REGION Network 14: таймер выключения частотника
   #tmrErrOffUZ(IN := NOT #qUZ AND #iWorkUZ, PT := #tStopPU_FC);   // TON
   IF #Ack OR #PU1.ack.%X5 THEN
       #errOff_UZ_PU1 := FALSE;   // RS flip-flop
   END_IF;
   IF #tmrErrOffUZ.Q THEN #errOff_UZ_PU1 := TRUE; END_IF;
   #PU1.st.%X5 := #errOff_UZ_PU1;
   IF #Ack OR #PU2.ack.%X5 THEN
       #errOff_UZ_PU2 := FALSE;   // RS flip-flop
   END_IF;
   IF #tmrErrOffUZ.Q THEN #errOff_UZ_PU2 := TRUE; END_IF;
   #PU2.st.%X5 := #errOff_UZ_PU2;
END_REGION

REGION Network 15: таймер включения контактора PU1
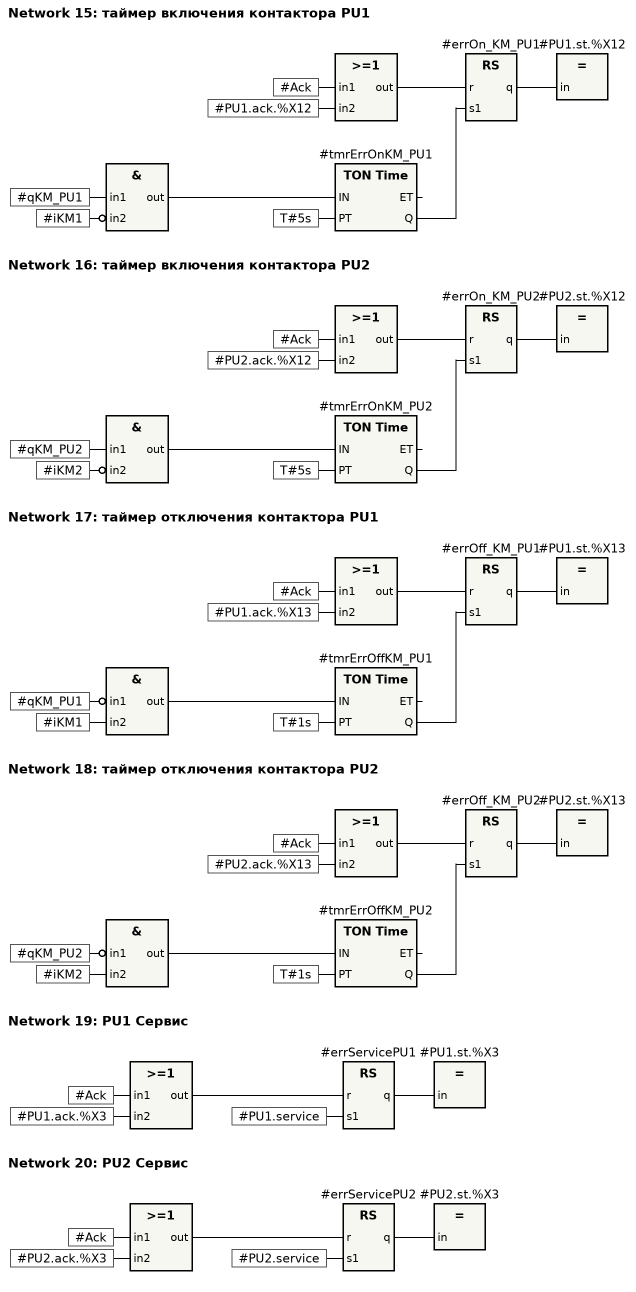
   #tmrErrOnKM_PU1(IN := #qKM_PU1 AND NOT #iKM1, PT := T#5s);   // TON
   IF #Ack OR #PU1.ack.%X12 THEN
       #errOn_KM_PU1 := FALSE;   // RS flip-flop
   END_IF;
   IF #tmrErrOnKM_PU1.Q THEN #errOn_KM_PU1 := TRUE; END_IF;
   #PU1.st.%X12 := #errOn_KM_PU1;
END_REGION

REGION Network 16: таймер включения контактора PU2
   #tmrErrOnKM_PU2(IN := #qKM_PU2 AND NOT #iKM2, PT := T#5s);   // TON
   IF #Ack OR #PU2.ack.%X12 THEN
       #errOn_KM_PU2 := FALSE;   // RS flip-flop
   END_IF;
   IF #tmrErrOnKM_PU2.Q THEN #errOn_KM_PU2 := TRUE; END_IF;
   #PU2.st.%X12 := #errOn_KM_PU2;
END_REGION

REGION Network 17: таймер отключения контактора PU1
   #tmrErrOffKM_PU1(IN := NOT #qKM_PU1 AND #iKM1, PT := T#1s);   // TON
   IF #Ack OR #PU1.ack.%X13 THEN
       #errOff_KM_PU1 := FALSE;   // RS flip-flop
   END_IF;
   IF #tmrErrOffKM_PU1.Q THEN #errOff_KM_PU1 := TRUE; END_IF;
   #PU1.st.%X13 := #errOff_KM_PU1;
END_REGION

REGION Network 18: таймер отключения контактора PU2
   #tmrErrOffKM_PU2(IN := NOT #qKM_PU2 AND #iKM2, PT := T#1s);   // TON
   IF #Ack OR #PU2.ack.%X13 THEN
       #errOff_KM_PU2 := FALSE;   // RS flip-flop
   END_IF;
   IF #tmrErrOffKM_PU2.Q THEN #errOff_KM_PU2 := TRUE; END_IF;
   #PU2.st.%X13 := #errOff_KM_PU2;
END_REGION

REGION Network 19: PU1 Сервис
   IF #Ack OR #PU1.ack.%X3 THEN
       #errServicePU1 := FALSE;   // RS flip-flop
   END_IF;
   IF #PU1.service THEN #errServicePU1 := TRUE; END_IF;
   #PU1.st.%X3 := #errServicePU1;
END_REGION

REGION Network 20: PU2 Сервис
   IF #Ack OR #PU2.ack.%X3 THEN
       #errServicePU2 := FALSE;   // RS flip-flop
   END_IF;
   IF #PU2.service THEN #errServicePU2 := TRUE; END_IF;
   #PU2.st.%X3 := #errServicePU2;
END_REGION

REGION Network 21: Сборная ошибка РU1
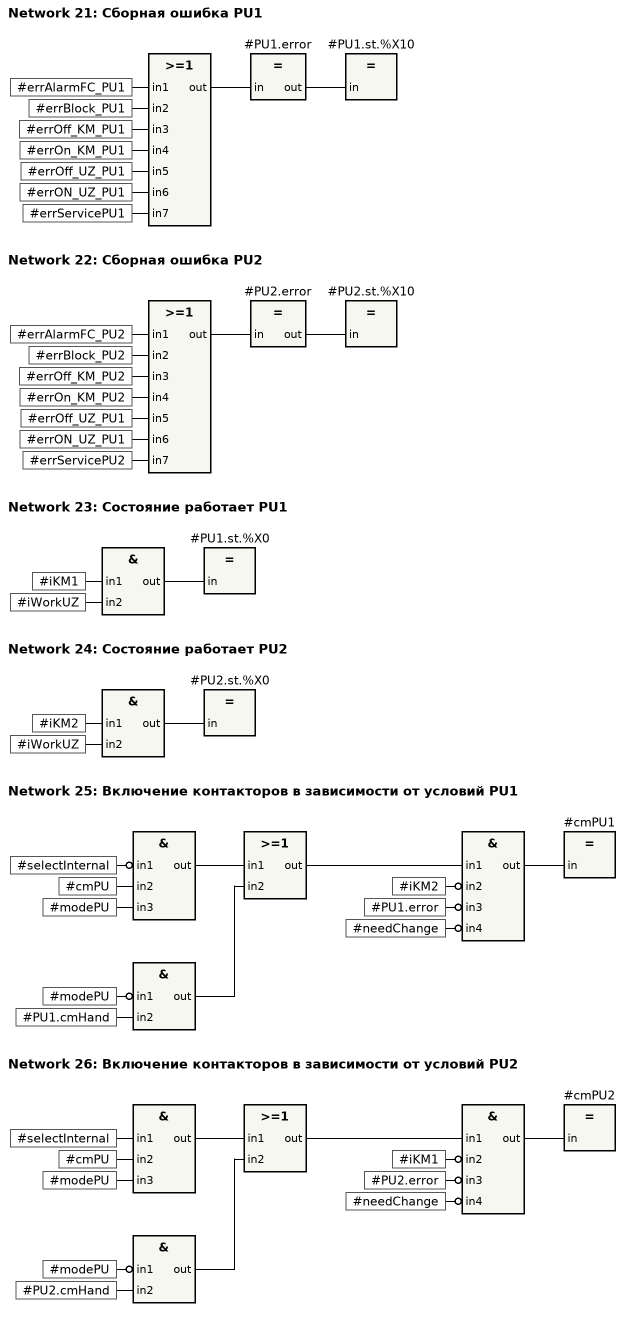
   #PU1.error := #errAlarmFC_PU1 OR #errBlock_PU1 OR #errOff_KM_PU1 OR #errOn_KM_PU1 OR #errOff_UZ_PU1 OR #errON_UZ_PU1 OR #errServicePU1;
   #PU1.st.%X10 := #PU1.error;
END_REGION

REGION Network 22: Сборная ошибка РU2
   #PU2.error := #errAlarmFC_PU2 OR #errBlock_PU2 OR #errOff_KM_PU2 OR #errOn_KM_PU2 OR #errOff_UZ_PU1 OR #errON_UZ_PU1 OR #errServicePU2;
   #PU2.st.%X10 := #PU2.error;
END_REGION

REGION Network 23: Состояние работает PU1
   #PU1.st.%X0 := #iKM1 AND #iWorkUZ;
END_REGION

REGION Network 24: Состояние работает PU2
   #PU2.st.%X0 := #iKM2 AND #iWorkUZ;
END_REGION

REGION Network 25: Включение контакторов в зависимости от условий PU1
   #cmPU1 := ((NOT #selectInternal AND #cmPU AND #modePU) OR (NOT #modePU AND #PU1.cmHand)) AND NOT #iKM2 AND NOT #PU1.error AND NOT #needChange;
END_REGION

REGION Network 26: Включение контакторов в зависимости от условий PU2
   #cmPU2 := ((#selectInternal AND #cmPU AND #modePU) OR (NOT #modePU AND #PU2.cmHand)) AND NOT #iKM1 AND NOT #PU2.error AND NOT #needChange;
END_REGION

REGION Network 27: Rонтактор первого насоса - СТОП
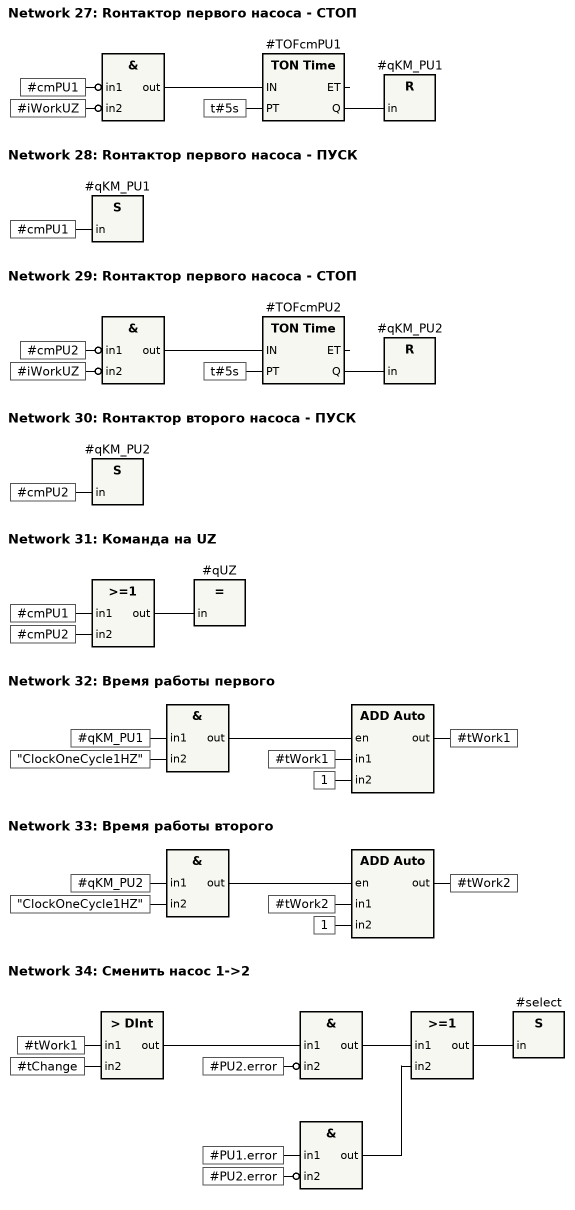
   #TOFcmPU1(IN := NOT #cmPU1 AND NOT #iWorkUZ, PT := t#5s);   // TON
   IF #TOFcmPU1.Q THEN #qKM_PU1 := FALSE; END_IF;
END_REGION

REGION Network 28: Rонтактор первого насоса - ПУСК
   IF #cmPU1 THEN #qKM_PU1 := TRUE; END_IF;
END_REGION

REGION Network 29: Rонтактор первого насоса - СТОП
   #TOFcmPU2(IN := NOT #cmPU2 AND NOT #iWorkUZ, PT := t#5s);   // TON
   IF #TOFcmPU2.Q THEN #qKM_PU2 := FALSE; END_IF;
END_REGION

REGION Network 30: Rонтактор второго насоса - ПУСК
   IF #cmPU2 THEN #qKM_PU2 := TRUE; END_IF;
END_REGION

REGION Network 31: Команда на UZ
   #qUZ := #cmPU1 OR #cmPU2;
END_REGION

REGION Network 32: Время работы первого
   IF #qKM_PU1 AND "ClockOneCycle1HZ" THEN #tWork1 := #tWork1 + 1; END_IF;
END_REGION

REGION Network 33: Время работы второго
   IF #qKM_PU2 AND "ClockOneCycle1HZ" THEN #tWork2 := #tWork2 + 1; END_IF;
END_REGION

REGION Network 34: Сменить насос 1->2
   IF ((#tWork1 > #tChange) AND NOT #PU2.error) OR (#PU1.error AND NOT #PU2.error) THEN
       #select := TRUE;
   END_IF;
END_REGION

REGION Network 35: Сменить насос 2->1
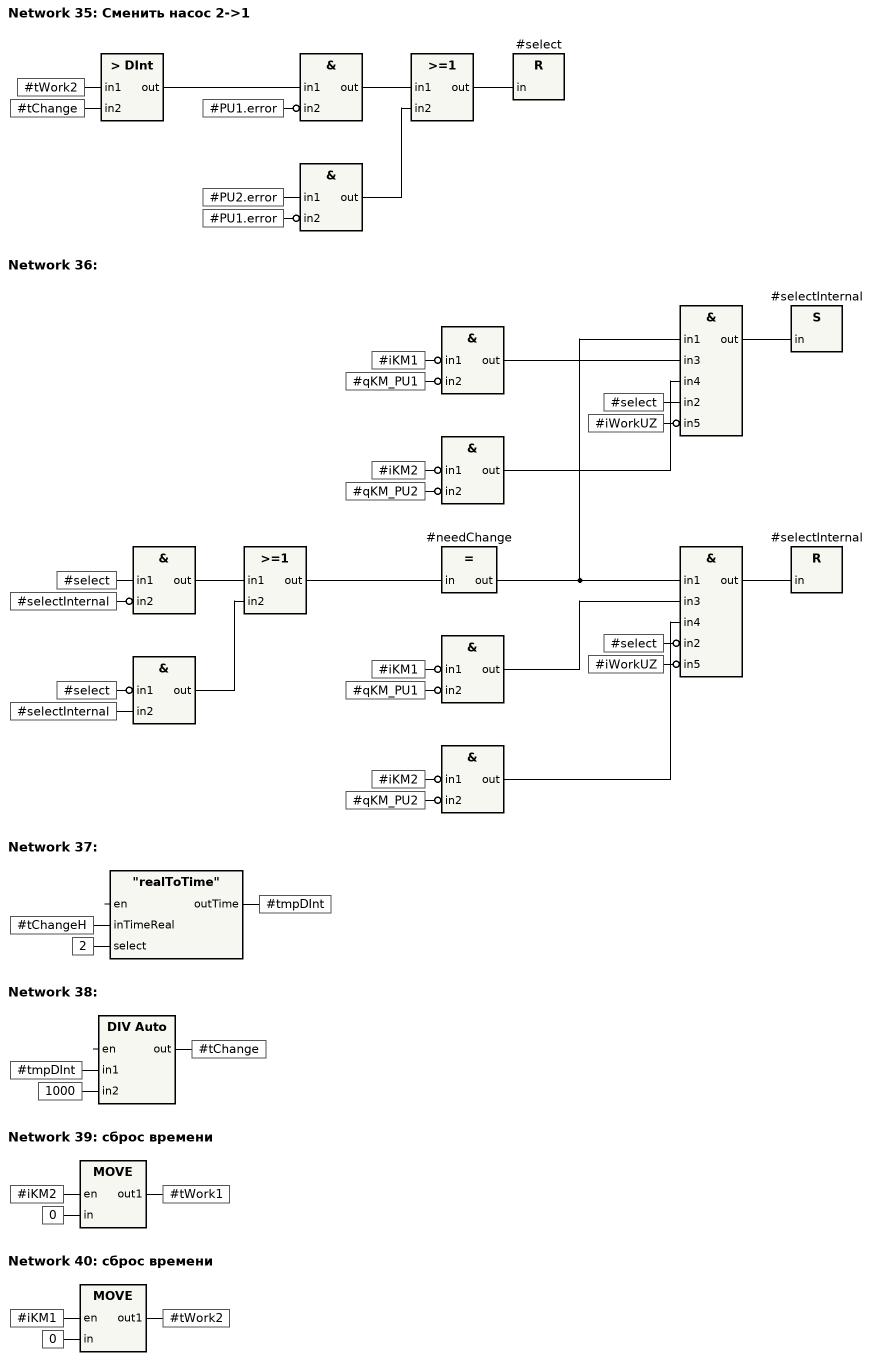
   IF ((#tWork2 > #tChange) AND NOT #PU1.error) OR (#PU2.error AND NOT #PU1.error) THEN
       #select := FALSE;
   END_IF;
END_REGION

REGION Network 36
   #needChange := (#select AND NOT #selectInternal) OR (NOT #select AND #selectInternal);
   IF #needChange AND NOT #iKM1 AND NOT #qKM_PU1 AND NOT #iKM2 AND NOT #qKM_PU2 AND #select AND NOT #iWorkUZ THEN
       #selectInternal := TRUE;
   END_IF;
   IF #needChange AND NOT #iKM1 AND NOT #qKM_PU1 AND NOT #iKM2 AND NOT #qKM_PU2 AND NOT #select AND NOT #iWorkUZ THEN
       #selectInternal := FALSE;
   END_IF;
END_REGION

REGION Network 37
   "realToTime"(inTimeReal := #tChangeH, select := 2, outTime => #tmpDInt);
END_REGION

REGION Network 38
   #tChange := #tmpDInt / 1000;
END_REGION

REGION Network 39: сброс времени
   IF #iKM2 THEN #tWork1 := 0; END_IF;
END_REGION

REGION Network 40: сброс времени
   IF #iKM1 THEN #tWork2 := 0; END_IF;
END_REGION

REGION Network 41: сброс ручных команд - PU1
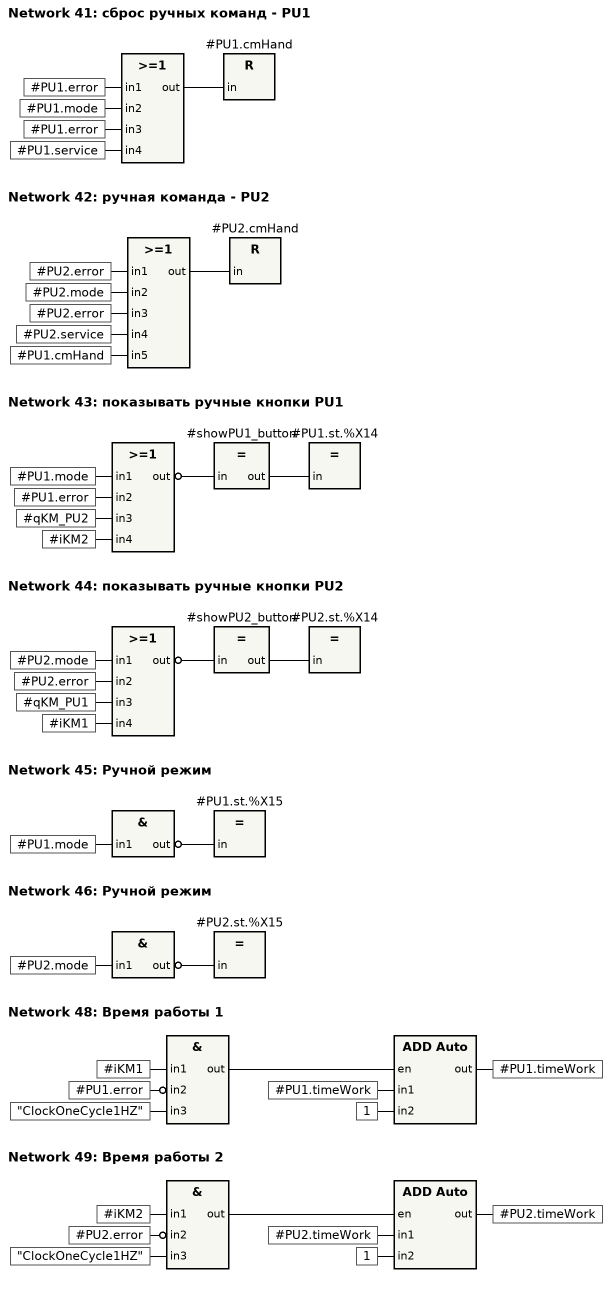
   IF #PU1.error OR #PU1.mode OR #PU1.error OR #PU1.service THEN #PU1.cmHand := FALSE; END_IF;
END_REGION

REGION Network 42: ручная команда - PU2
   IF #PU2.error OR #PU2.mode OR #PU2.error OR #PU2.service OR #PU1.cmHand THEN #PU2.cmHand := FALSE; END_IF;
END_REGION

REGION Network 43: показывать ручные кнопки PU1
   #showPU1_button := NOT (#PU1.mode OR #PU1.error OR #qKM_PU2 OR #iKM2);
   #PU1.st.%X14 := #showPU1_button;
END_REGION

REGION Network 44: показывать ручные кнопки PU2
   #showPU2_button := NOT (#PU2.mode OR #PU2.error OR #qKM_PU1 OR #iKM1);
   #PU2.st.%X14 := #showPU2_button;
END_REGION

REGION Network 45: Ручной режим
   #PU1.st.%X15 := NOT #PU1.mode;
END_REGION

REGION Network 46: Ручной режим
   #PU2.st.%X15 := NOT #PU2.mode;
END_REGION

REGION Network 47 (SCL): Сброс битов Ack
   IF NOT #PU1.st.%X0 AND #PU1.ack.%X0 THEN
       #PU1.ack.%X0 := 0;
   END_IF;
   IF NOT #PU1.st.%X1 AND #PU1.ack.%X1 THEN
       #PU1.ack.%X1 := 0;
   END_IF;
   IF NOT #PU1.st.%X2 AND #PU1.ack.%X2 THEN
       #PU1.ack.%X2 := 0;
   END_IF;
   IF NOT #PU1.st.%X3 AND #PU1.ack.%X3 THEN
       #PU1.ack.%X3 := 0;
   END_IF;
   IF NOT #PU1.st.%X4 AND #PU1.ack.%X4 THEN
       #PU1.ack.%X4 := 0;
   END_IF;
   IF NOT #PU1.st.%X5 AND #PU1.ack.%X5 THEN
       #PU1.ack.%X5 := 0;
   END_IF;
   IF NOT #PU1.st.%X6 AND #PU1.ack.%X6 THEN
       #PU1.ack.%X6 := 0;
   END_IF;
   IF NOT #PU1.st.%X7 AND #PU1.ack.%X7 THEN
       #PU1.ack.%X7 := 0;
   END_IF;
   IF NOT #PU1.st.%X8 AND #PU1.ack.%X8 THEN
       #PU1.ack.%X8 := 0;
   END_IF;
   IF NOT #PU1.st.%X9 AND #PU1.ack.%X9 THEN
       #PU1.ack.%X9 := 0;
   END_IF;
   IF NOT #PU1.st.%X10 AND #PU1.ack.%X10 THEN
       #PU1.ack.%X10 := 0;
   END_IF;
   IF NOT #PU1.st.%X11 AND #PU1.ack.%X11 THEN
       #PU1.ack.%X11 := 0;
   END_IF;
   IF NOT #PU1.st.%X12 AND #PU1.ack.%X12 THEN
       #PU1.ack.%X12 := 0;
   END_IF;
   IF NOT #PU1.st.%X13 AND #PU1.ack.%X13 THEN
       #PU1.ack.%X13 := 0;
   END_IF;
   IF NOT #PU1.st.%X14 AND #PU1.ack.%X14 THEN
       #PU1.ack.%X14 := 0;
   END_IF;
   IF NOT #PU1.st.%X15 AND #PU1.ack.%X15 THEN
       #PU1.ack.%X15 := 0;
   END_IF;
   IF NOT #PU2.st.%X0 AND #PU2.ack.%X0 THEN
       #PU2.ack.%X0 := 0;
   END_IF;
   IF NOT #PU2.st.%X1 AND #PU2.ack.%X1 THEN
       #PU2.ack.%X1 := 0;
   END_IF;
   IF NOT #PU2.st.%X2 AND #PU2.ack.%X2 THEN
       #PU2.ack.%X2 := 0;
   END_IF;
   IF NOT #PU2.st.%X3 AND #PU2.ack.%X3 THEN
       #PU2.ack.%X3 := 0;
   END_IF;
   IF NOT #PU2.st.%X4 AND #PU2.ack.%X4 THEN
       #PU2.ack.%X4 := 0;
   END_IF;
   IF NOT #PU2.st.%X5 AND #PU2.ack.%X5 THEN
       #PU2.ack.%X5 := 0;
   END_IF;
   IF NOT #PU2.st.%X6 AND #PU2.ack.%X6 THEN
       #PU2.ack.%X6 := 0;
   END_IF;
   IF NOT #PU2.st.%X7 AND #PU2.ack.%X7 THEN
       #PU2.ack.%X7 := 0;
   END_IF;
   IF NOT #PU2.st.%X8 AND #PU2.ack.%X8 THEN
       #PU2.ack.%X8 := 0;
   END_IF;
   IF NOT #PU2.st.%X9 AND #PU2.ack.%X9 THEN
       #PU2.ack.%X9 := 0;
   END_IF;
   IF NOT #PU2.st.%X10 AND #PU2.ack.%X10 THEN
       #PU2.ack.%X10 := 0;
   END_IF;
   IF NOT #PU2.st.%X11 AND #PU2.ack.%X11 THEN
       #PU2.ack.%X11 := 0;
   END_IF;
   IF NOT #PU2.st.%X12 AND #PU2.ack.%X12 THEN
       #PU2.ack.%X12 := 0;
   END_IF;
   IF NOT #PU2.st.%X13 AND #PU2.ack.%X13 THEN
       #PU2.ack.%X13 := 0;
   END_IF;
   IF NOT #PU2.st.%X14 AND #PU2.ack.%X14 THEN
       #PU2.ack.%X14 := 0;
   END_IF;
   IF NOT #PU2.st.%X15 AND #PU2.ack.%X15 THEN
       #PU2.ack.%X15 := 0;
   END_IF;
END_REGION

REGION Network 48: Время работы 1
   IF #iKM1 AND NOT #PU1.error AND "ClockOneCycle1HZ" THEN #PU1.timeWork := #PU1.timeWork + 1; END_IF;
END_REGION

REGION Network 49: Время работы 2
   IF #iKM2 AND NOT #PU2.error AND "ClockOneCycle1HZ" THEN #PU2.timeWork := #PU2.timeWork + 1; END_IF;
END_REGION

REGION Network 50: Сброс 1
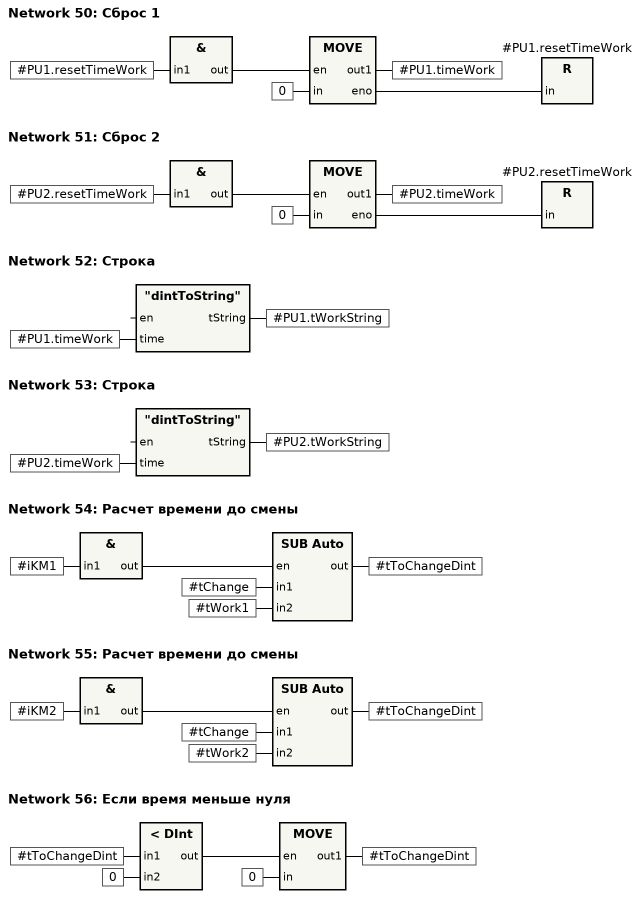
   IF #PU1.resetTimeWork THEN
       #PU1.timeWork := 0;
       #PU1.resetTimeWork := FALSE;
   END_IF;
END_REGION

REGION Network 51: Сброс 2
   IF #PU2.resetTimeWork THEN
       #PU2.timeWork := 0;
       #PU2.resetTimeWork := FALSE;
   END_IF;
END_REGION

REGION Network 52: Строка
   "dintToString"("time" := #PU1.timeWork, tString => #PU1.tWorkString);
END_REGION

REGION Network 53: Строка
   "dintToString"("time" := #PU2.timeWork, tString => #PU2.tWorkString);
END_REGION

REGION Network 54: Расчет времени до смены
   IF #iKM1 THEN #tToChangeDint := #tChange - #tWork1; END_IF;
END_REGION

REGION Network 55: Расчет времени до смены
   IF #iKM2 THEN #tToChangeDint := #tChange - #tWork2; END_IF;
END_REGION

REGION Network 56: Если время меньше нуля
   IF #tToChangeDint < 0 THEN #tToChangeDint := 0; END_IF;
END_REGION

REGION Network 57 (SCL): Сек -> час
   #tToChangeRealHour := DINT_TO_REAL(#tToChangeDint) / 3600.0;
END_REGION
END_FUNCTION_BLOCK

FUNCTION "intToTime" : Void
{ S7_Optimized_Access := 'TRUE' }
VERSION : 0.1
   VAR_INPUT 
      intTime : Int;
      select : Int;   // 0-sec, 1-min,2-hour
   END_VAR

   VAR_OUTPUT 
      tOut : Time;
   END_VAR


BEGIN
	CASE #select OF
	    0:
	        #tOut := DINT_TO_TIME(INT_TO_DINT(#intTime) * 1000);
	    1:
	        #tOut := DINT_TO_TIME(INT_TO_DINT(#intTime)* 60000);
	    2:
	        #tOut := DINT_TO_TIME(INT_TO_DINT(#intTime) * 3600000);
	    ELSE  // Statement section ELSE
	        #tOut := t#0s;
	END_CASE;
END_FUNCTION

FUNCTION "bitToWord" : Void   // FC5, LAD
{ S7_Optimized_Access := 'TRUE' }
VERSION : 0.1
// stored: AutoNumber true, IsIECCheckEnabled false, SetENOAutomatically false, UDAEnableTagReadback false
   VAR_INPUT
      inBit0 : Bool;
      inBit1 : Bool;
      inBit2 : Bool;
      inBit3 : Bool;
      inBit4 : Bool;
      inBit5 : Bool;
      inBit6 : Bool;
      inBit7 : Bool;
      inBit8 : Bool;
      inBit9 : Bool;
      inBit10 : Bool;
      inBit11 : Bool;
      inBit12 : Bool;
      inBit13 : Bool;
      inBit14 : Bool;
      inBit15 : Bool;
   END_VAR
   VAR_OUTPUT
      outWord : Word;
   END_VAR
BEGIN

REGION Network 1
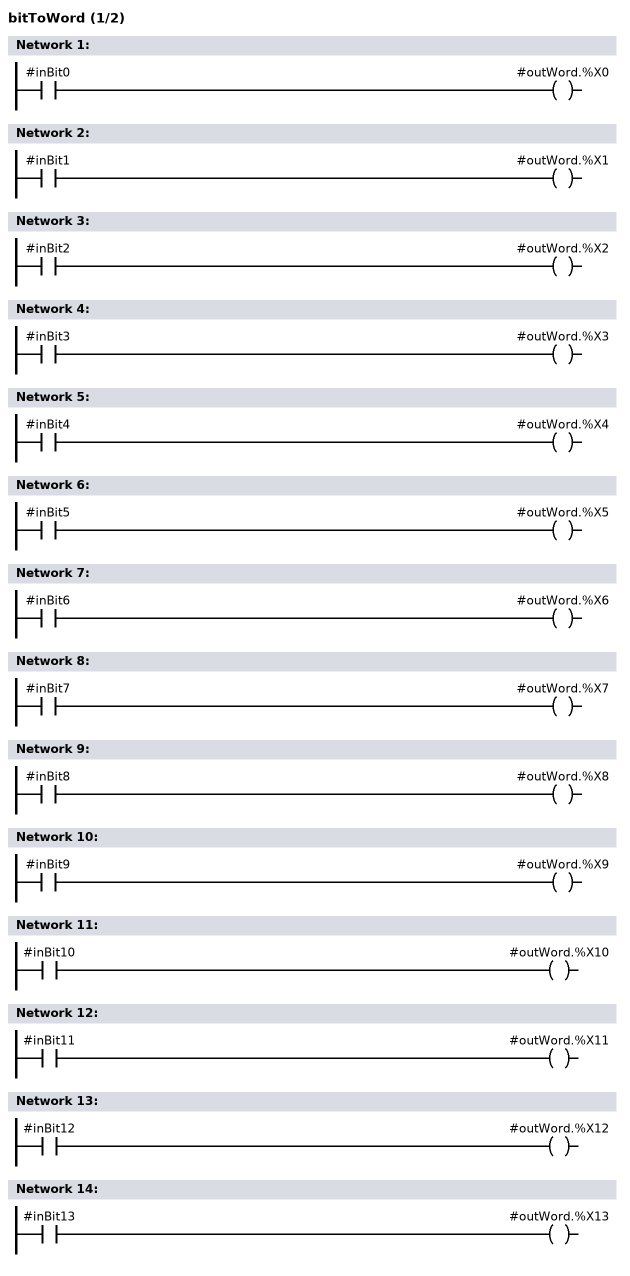
   RUNG wire#powerrail
      Contact( #inBit0 )
      Coil( #outWord.%X0 )
   END_RUNG
   // the same network as SCL:
   #outWord.%X0 := #inBit0;
END_REGION

REGION Network 2
   RUNG wire#powerrail
      Contact( #inBit1 )
      Coil( #outWord.%X1 )
   END_RUNG
   // the same network as SCL:
   #outWord.%X1 := #inBit1;
END_REGION

REGION Network 3
   RUNG wire#powerrail
      Contact( #inBit2 )
      Coil( #outWord.%X2 )
   END_RUNG
   // the same network as SCL:
   #outWord.%X2 := #inBit2;
END_REGION

REGION Network 4
   RUNG wire#powerrail
      Contact( #inBit3 )
      Coil( #outWord.%X3 )
   END_RUNG
   // the same network as SCL:
   #outWord.%X3 := #inBit3;
END_REGION

REGION Network 5
   RUNG wire#powerrail
      Contact( #inBit4 )
      Coil( #outWord.%X4 )
   END_RUNG
   // the same network as SCL:
   #outWord.%X4 := #inBit4;
END_REGION

REGION Network 6
   RUNG wire#powerrail
      Contact( #inBit5 )
      Coil( #outWord.%X5 )
   END_RUNG
   // the same network as SCL:
   #outWord.%X5 := #inBit5;
END_REGION

REGION Network 7
   RUNG wire#powerrail
      Contact( #inBit6 )
      Coil( #outWord.%X6 )
   END_RUNG
   // the same network as SCL:
   #outWord.%X6 := #inBit6;
END_REGION

REGION Network 8
   RUNG wire#powerrail
      Contact( #inBit7 )
      Coil( #outWord.%X7 )
   END_RUNG
   // the same network as SCL:
   #outWord.%X7 := #inBit7;
END_REGION

REGION Network 9
   RUNG wire#powerrail
      Contact( #inBit8 )
      Coil( #outWord.%X8 )
   END_RUNG
   // the same network as SCL:
   #outWord.%X8 := #inBit8;
END_REGION

REGION Network 10
   RUNG wire#powerrail
      Contact( #inBit9 )
      Coil( #outWord.%X9 )
   END_RUNG
   // the same network as SCL:
   #outWord.%X9 := #inBit9;
END_REGION

REGION Network 11
   RUNG wire#powerrail
      Contact( #inBit10 )
      Coil( #outWord.%X10 )
   END_RUNG
   // the same network as SCL:
   #outWord.%X10 := #inBit10;
END_REGION

REGION Network 12
   RUNG wire#powerrail
      Contact( #inBit11 )
      Coil( #outWord.%X11 )
   END_RUNG
   // the same network as SCL:
   #outWord.%X11 := #inBit11;
END_REGION

REGION Network 13
   RUNG wire#powerrail
      Contact( #inBit12 )
      Coil( #outWord.%X12 )
   END_RUNG
   // the same network as SCL:
   #outWord.%X12 := #inBit12;
END_REGION

REGION Network 14
   RUNG wire#powerrail
      Contact( #inBit13 )
      Coil( #outWord.%X13 )
   END_RUNG
   // the same network as SCL:
   #outWord.%X13 := #inBit13;
END_REGION

REGION Network 15
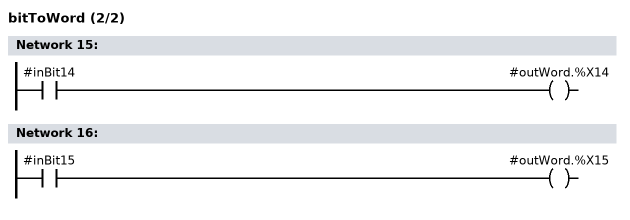
   RUNG wire#powerrail
      Contact( #inBit14 )
      Coil( #outWord.%X14 )
   END_RUNG
   // the same network as SCL:
   #outWord.%X14 := #inBit14;
END_REGION

REGION Network 16
   RUNG wire#powerrail
      Contact( #inBit15 )
      Coil( #outWord.%X15 )
   END_RUNG
   // the same network as SCL:
   #outWord.%X15 := #inBit15;
END_REGION
END_FUNCTION

FUNCTION "realToTime" : Void
{ S7_Optimized_Access := 'TRUE' }
VERSION : 0.1
   VAR_INPUT 
      inTimeReal : Real;
      select : Int;   // 0-секунды, 1-минуты, 2-часы
   END_VAR

   VAR_OUTPUT 
      outTime : Time;
   END_VAR


BEGIN
	CASE #select OF
	    0:
	        #outTime := DINT_TO_TIME(REAL_TO_DINT(#inTimeReal * 1000.0));
	    1:
	        #outTime := DINT_TO_TIME(REAL_TO_DINT(#inTimeReal * 60000.0));
	    2:
	        #outTime := DINT_TO_TIME(REAL_TO_DINT(#inTimeReal * 1000.0) * 3600);
	    ELSE  // Statement section ELSE
	        #outTime := t#0s;
	END_CASE;
	
END_FUNCTION

FUNCTION "dintToString" : Void
{ S7_Optimized_Access := 'TRUE' }
VERSION : 0.1
   VAR_INPUT 
      "time" : UDInt;
   END_VAR

   VAR_OUTPUT 
      tString : String;
   END_VAR

   VAR_TEMP 
      tDInt : UDInt;
      size : USInt;
      pos : USInt;
      day : DInt;
      h : DInt;
      m : DInt;
      s : DInt;
   END_VAR


BEGIN
	#tDInt := #time;
	
	//сбор строки
	#day := #tDInt / 86400;
	#h := (#tDInt MOD 86400) / 3600;
	#m := (#tDInt MOD 3600) / 60;
	#s := #tDInt MOD 60;
	#tString := '00000:00:00:00';
	
	VAL_STRG(IN := #day,
	         SIZE := 5,
	         PREC := 0,
	         FORMAT := 1,
	         P := 1,
	         OUT => #tString);
	
	IF #h < 10 THEN
	    #size := 1;
	    #pos := 8;
	ELSE
	    #size := 2;
	    #pos := 7;
	END_IF;
	
	VAL_STRG(IN := #h,
	         SIZE := #size,
	         PREC := 0,
	         FORMAT := 1,
	         P := #pos,
	         OUT => #tString);
	
	IF #m < 10 THEN
	    #size := 1;
	    #pos := 11;
	ELSE
	    #size := 2;
	    #pos := 10;
	END_IF;
	
	VAL_STRG(IN := #m,
	         SIZE := #size,
	         PREC := 0,
	         FORMAT := 1,
	         P := #pos,
	         OUT => #tString);
	IF #s < 10 THEN
	    #size := 1;
	    #pos := 14;
	ELSE
	    #size := 2;
	    #pos := 13;
	END_IF;
	VAL_STRG(IN := #s,
	         SIZE := #size,
	         PREC := 0,
	         FORMAT := 1,
	         P := #pos,
	         OUT => #tString);
END_FUNCTION

FUNCTION_BLOCK "noPulseTOF"   // FB15, FBD
{ S7_Optimized_Access := 'TRUE' }
VERSION : 0.1
// stored: AutoNumber true, IsIECCheckEnabled false, IsRetainMemResEnabled false, MemoryReserve 100, SetENOAutomatically false, UDAEnableTagReadback false
   VAR_INPUT
      pulse : Bool;
      timeSP_sec : Real;
      reset : Bool;
   END_VAR
   VAR_OUTPUT
      out : Bool;
   END_VAR
   VAR
      curTime : Real;
      nTrig : Bool;
      pTirg : Bool;
   END_VAR
   VAR_TEMP   // added for the SCL form of the ladder/FBD networks
      _w1 : Bool;
      _w2 : Bool;
   END_VAR
BEGIN

REGION Network 1: Увеличение времени
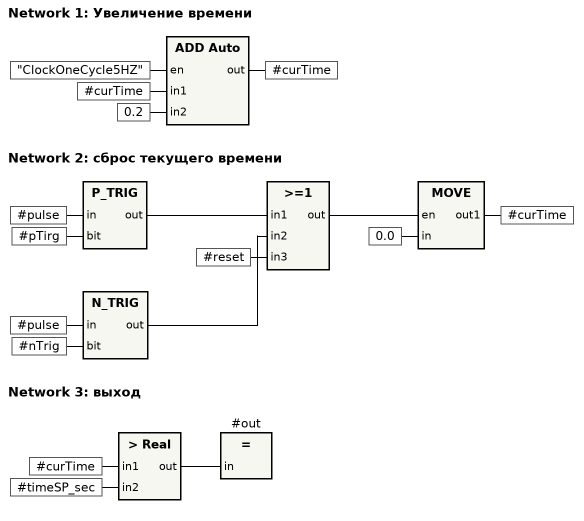
   IF "ClockOneCycle5HZ" THEN #curTime := #curTime + 0.2; END_IF;
END_REGION

REGION Network 2: сброс текущего времени
   #_w1 := #pulse AND NOT #pTirg;   // rising edge
   #pTirg := #pulse;
   #_w2 := NOT #pulse AND #nTrig;   // falling edge
   #nTrig := #pulse;
   IF #_w1 OR #_w2 OR #reset THEN #curTime := 0.0; END_IF;
END_REGION

REGION Network 3: выход
   #out := #curTime > #timeSP_sec;
END_REGION
END_FUNCTION_BLOCK

FUNCTION_BLOCK "sel2pu"   // FB4, FBD
{ S7_Optimized_Access := 'TRUE' }
VERSION : 0.1
// stored: AutoNumber true, IsIECCheckEnabled false, IsRetainMemResEnabled false, MemoryReserve 100, SetENOAutomatically false, UDAEnableTagReadback false
   VAR_INPUT
      cmStart : Bool;
      mode : Bool;
      tChangeHReal : Real;
   END_VAR
   VAR_OUTPUT
      tToChange : Real;
   END_VAR
   VAR_IN_OUT
      PU1 : "Pump";
      PU2 : "Pump";
      select : Bool;
   END_VAR
   VAR
      tWork1 : DInt;
      tWork2 : DInt;
      tChangeDInt : DInt;
   END_VAR
BEGIN

REGION Network 1: Режим работы
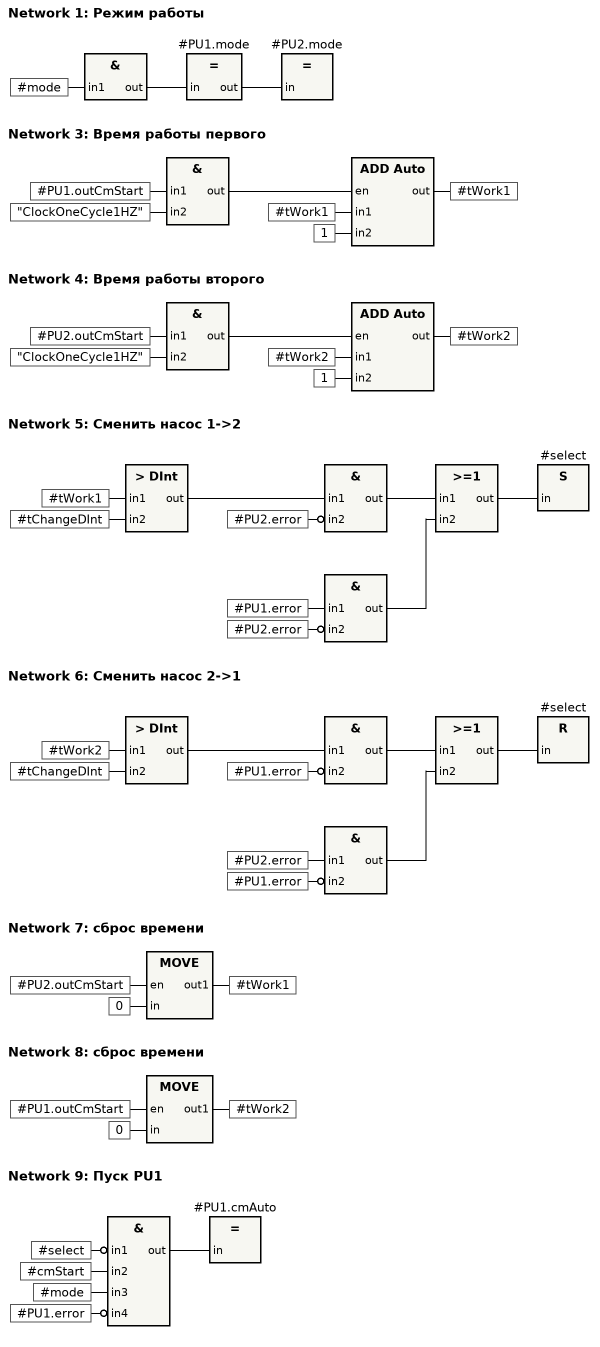
   #PU1.mode := #mode;
   #PU2.mode := #mode;
END_REGION

REGION Network 2 (SCL): Преобразование времен
   #tChangeDInt := REAL_TO_DINT(#tChangeHReal * 3600.0);
END_REGION

REGION Network 3: Время работы первого
   IF #PU1.outCmStart AND "ClockOneCycle1HZ" THEN #tWork1 := #tWork1 + 1; END_IF;
END_REGION

REGION Network 4: Время работы второго
   IF #PU2.outCmStart AND "ClockOneCycle1HZ" THEN #tWork2 := #tWork2 + 1; END_IF;
END_REGION

REGION Network 5: Сменить насос 1->2
   IF ((#tWork1 > #tChangeDInt) AND NOT #PU2.error) OR (#PU1.error AND NOT #PU2.error) THEN
       #select := TRUE;
   END_IF;
END_REGION

REGION Network 6: Сменить насос 2->1
   IF ((#tWork2 > #tChangeDInt) AND NOT #PU1.error) OR (#PU2.error AND NOT #PU1.error) THEN
       #select := FALSE;
   END_IF;
END_REGION

REGION Network 7: сброс времени
   IF #PU2.outCmStart THEN #tWork1 := 0; END_IF;
END_REGION

REGION Network 8: сброс времени
   IF #PU1.outCmStart THEN #tWork2 := 0; END_IF;
END_REGION

REGION Network 9: Пуск PU1
   #PU1.cmAuto := NOT #select AND #cmStart AND #mode AND NOT #PU1.error;
END_REGION

REGION Network 10: Пуск PU2
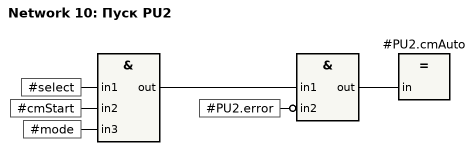
   #PU2.cmAuto := #select AND #cmStart AND #mode AND NOT #PU2.error;
END_REGION
END_FUNCTION_BLOCK

FUNCTION_BLOCK "PumpCntr"   // FB60, LAD
{ S7_Optimized_Access := 'FALSE' }
VERSION : 0.1
// #ST:
// номер бита, часло десятичное
//  0  - стоп 
// 0 1 - работа
// 1 2 - запуск
// 2 4 - остановка
// 3 8 - сервисный режим
// 4 16 - ошибка Пуска
// 5 32 - ошибка Стопа
// 6 64 - ошибка питания
// 7 128 - ошибка частотника (дозатора)
// 8 256 - Блокировка внешняя
// 9 - 512 - нажат аварийный стоп
// 10 -1024 - сборная авария
// 11 2048 - местный режим
// 12 4096
// 13 8192
// 14 16384 1-показывать кнопки ручного управления
// 15 32768 - режим 1-ручной, 0-авто (только для индкатора на скаде)
// stored: AutoNumber false, IsIECCheckEnabled false, SetENOAutomatically false, UDAEnableTagReadback false
   VAR_INPUT
      power : Bool;   // питание устройства 1-ок
      run : Bool;   // 1-работа
      emrStop : Bool;   // Авариный стоп 0-авария, 1-ок
      local : Bool;   // 1-местный режим
      alarmFC : Bool;   // 1-авария
      block1 : Bool;
      block2 : Bool;
      block3 : Bool;
      block4 : Bool;
      block5 : Bool;
      block6 : Bool;
      block7 : Bool;
      block8 : Bool;
   END_VAR
   VAR_OUTPUT
      qStart : Bool;   // пуск
   END_VAR
   VAR_IN_OUT
      dev : "Pump";
   END_VAR
   VAR DB_SPECIFIC
      ErrOC : Bool;   // Признак аварии по закрытию или открытию
      ErrPower : Bool;   // Признак аварии питания
      ErrDis : Bool;   // Признак внешней блокировки
      qON : Bool;   // Выход для управления механизмом
      tmrClosing { S7_SetPoint := 'True'} : TON_TIME;
      tmrOpening { S7_SetPoint := 'True'} : TON_TIME;
      closed : Bool;
      opened : Bool;
      closing : Bool;
      opening : Bool;
      errStart : Bool;
      errStop : Bool;
      errEmrStop : Bool;
      errAlarmFc : Bool;
      errService : Bool;
      errLocal : Bool;
      tStart : Time;
      tStop : Time;
   END_VAR
   VAR
      DpumpAckAlarm_Instance : "PumpAckAlarm";
   END_VAR
   VAR CONSTANT
      ACK_DELAY : Time := T#1s;
   END_VAR
BEGIN

REGION Network 1: Сброс состояния
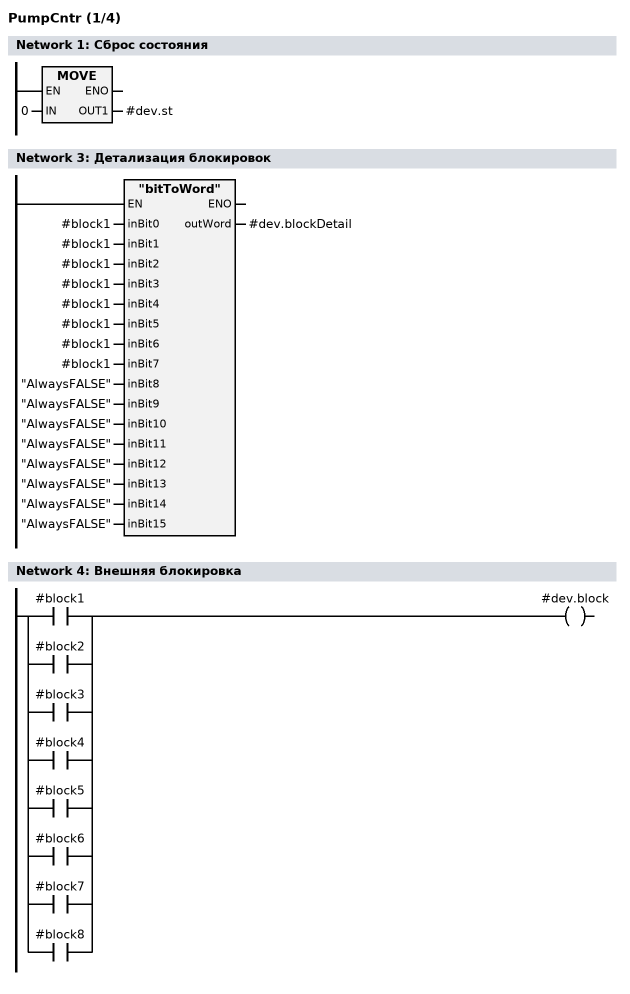
   RUNG wire#powerrail
      { S7_GenerateENO := "TRUE" } Move(in := 0, out1 => #dev.st)
   END_RUNG
   // the same network as SCL:
   #dev.st := 0;
END_REGION

REGION Network 3: Детализация блокировок
   RUNG wire#powerrail
      "bitToWord"(inBit0 := #block1, inBit1 := #block1, inBit2 := #block1, inBit3 := #block1, inBit4 := #block1, inBit5 := #block1, inBit6 := #block1, inBit7 := #block1, inBit8 := "AlwaysFALSE", inBit9 := "AlwaysFALSE", inBit10 := "AlwaysFALSE", inBit11 := "AlwaysFALSE", inBit12 := "AlwaysFALSE", inBit13 := "AlwaysFALSE", inBit14 := "AlwaysFALSE", inBit15 := "AlwaysFALSE", outWord => #dev.blockDetail)
   END_RUNG
   // the same network as SCL:
   "bitToWord"(inBit0 := #block1,
               inBit1 := #block1,
               inBit2 := #block1,
               inBit3 := #block1,
               inBit4 := #block1,
               inBit5 := #block1,
               inBit6 := #block1,
               inBit7 := #block1,
               inBit8 := "AlwaysFALSE",
               inBit9 := "AlwaysFALSE",
               inBit10 := "AlwaysFALSE",
               inBit11 := "AlwaysFALSE",
               inBit12 := "AlwaysFALSE",
               inBit13 := "AlwaysFALSE",
               inBit14 := "AlwaysFALSE",
               inBit15 := "AlwaysFALSE",
               outWord => #dev.blockDetail);
END_REGION

REGION Network 4: Внешняя блокировка
   RUNG wire#powerrail
      Contact( #block1 )
      wire#w1
      Coil( #dev.block )
   END_RUNG
   RUNG wire#powerrail
      Contact( #block2 )
   END_RUNG wire#w1
   RUNG wire#powerrail
      Contact( #block3 )
   END_RUNG wire#w1
   RUNG wire#powerrail
      Contact( #block4 )
   END_RUNG wire#w1
   RUNG wire#powerrail
      Contact( #block5 )
   END_RUNG wire#w1
   RUNG wire#powerrail
      Contact( #block6 )
   END_RUNG wire#w1
   RUNG wire#powerrail
      Contact( #block7 )
   END_RUNG wire#w1
   RUNG wire#powerrail
      Contact( #block8 )
   END_RUNG wire#w1
   // the same network as SCL:
   #dev.block := #block1 OR #block2 OR #block3 OR #block4 OR #block5 OR #block6 OR #block7 OR #block8;
END_REGION

REGION Network 5: Alarms
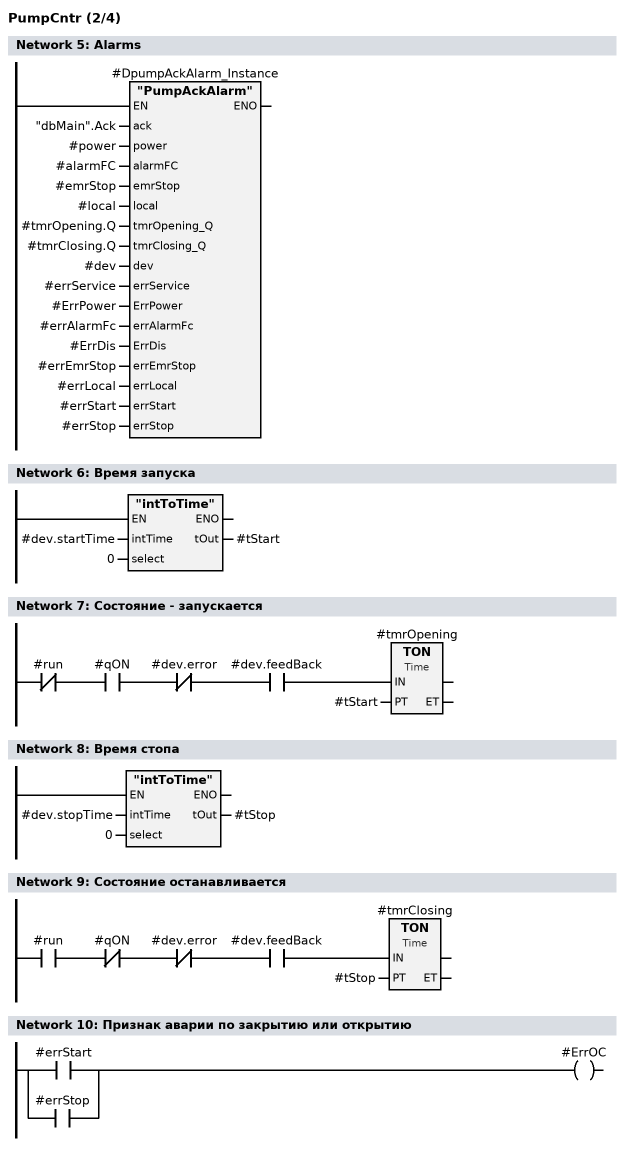
   RUNG wire#powerrail
      #DpumpAckAlarm_Instance(ack := "dbMain".Ack, power := #power, alarmFC := #alarmFC, emrStop := #emrStop, local := #local, tmrOpening_Q := #tmrOpening.Q, tmrClosing_Q := #tmrClosing.Q, dev := #dev, errService := #errService, ErrPower := #ErrPower, errAlarmFc := #errAlarmFc, ErrDis := #ErrDis, errEmrStop := #errEmrStop, errLocal := #errLocal, errStart := #errStart, errStop := #errStop)
   END_RUNG
   // the same network as SCL:
   #DpumpAckAlarm_Instance(ack := "dbMain".Ack,   // "PumpAckAlarm"
                           power := #power,
                           alarmFC := #alarmFC,
                           emrStop := #emrStop,
                           local := #local,
                           tmrOpening_Q := #tmrOpening.Q,
                           tmrClosing_Q := #tmrClosing.Q,
                           dev := #dev,
                           errService := #errService,
                           ErrPower := #ErrPower,
                           errAlarmFc := #errAlarmFc,
                           ErrDis := #ErrDis,
                           errEmrStop := #errEmrStop,
                           errLocal := #errLocal,
                           errStart := #errStart,
                           errStop := #errStop);
END_REGION

REGION Network 6: Время запуска
   RUNG wire#powerrail
      "intToTime"(intTime := #dev.startTime, select := 0, tOut => #tStart)
   END_RUNG
   // the same network as SCL:
   "intToTime"(intTime := #dev.startTime, select := 0, tOut => #tStart);
END_REGION

REGION Network 7: Состояние - запускается
   RUNG wire#powerrail
      I_Contact( #run )
      Contact( #qON )
      I_Contact( #dev.error )
      Contact( #dev.feedBack )
      { S7_Templates := "time_type := Time" } #tmrOpening.TON(pt := #tStart, et =>)
   END_RUNG
   // the same network as SCL:
   #tmrOpening(IN := NOT #run AND #qON AND NOT #dev.error AND #dev.feedBack, PT := #tStart);   // TON
END_REGION

REGION Network 8: Время стопа
   RUNG wire#powerrail
      "intToTime"(intTime := #dev.stopTime, select := 0, tOut => #tStop)
   END_RUNG
   // the same network as SCL:
   "intToTime"(intTime := #dev.stopTime, select := 0, tOut => #tStop);
END_REGION

REGION Network 9: Состояние останавливается
   RUNG wire#powerrail
      Contact( #run )
      I_Contact( #qON )
      I_Contact( #dev.error )
      Contact( #dev.feedBack )
      { S7_Templates := "time_type := Time" } #tmrClosing.TON(pt := #tStop, et =>)
   END_RUNG
   // the same network as SCL:
   #tmrClosing(IN := #run AND NOT #qON AND NOT #dev.error AND #dev.feedBack, PT := #tStop);   // TON
END_REGION

REGION Network 10: Признак аварии по закрытию или открытию
   RUNG wire#powerrail
      Contact( #errStart )
      wire#w1
      Coil( #ErrOC )
   END_RUNG
   RUNG wire#powerrail
      Contact( #errStop )
   END_RUNG wire#w1
   // the same network as SCL:
   #ErrOC := #errStart OR #errStop;
END_REGION

REGION Network 11: Сборная авария
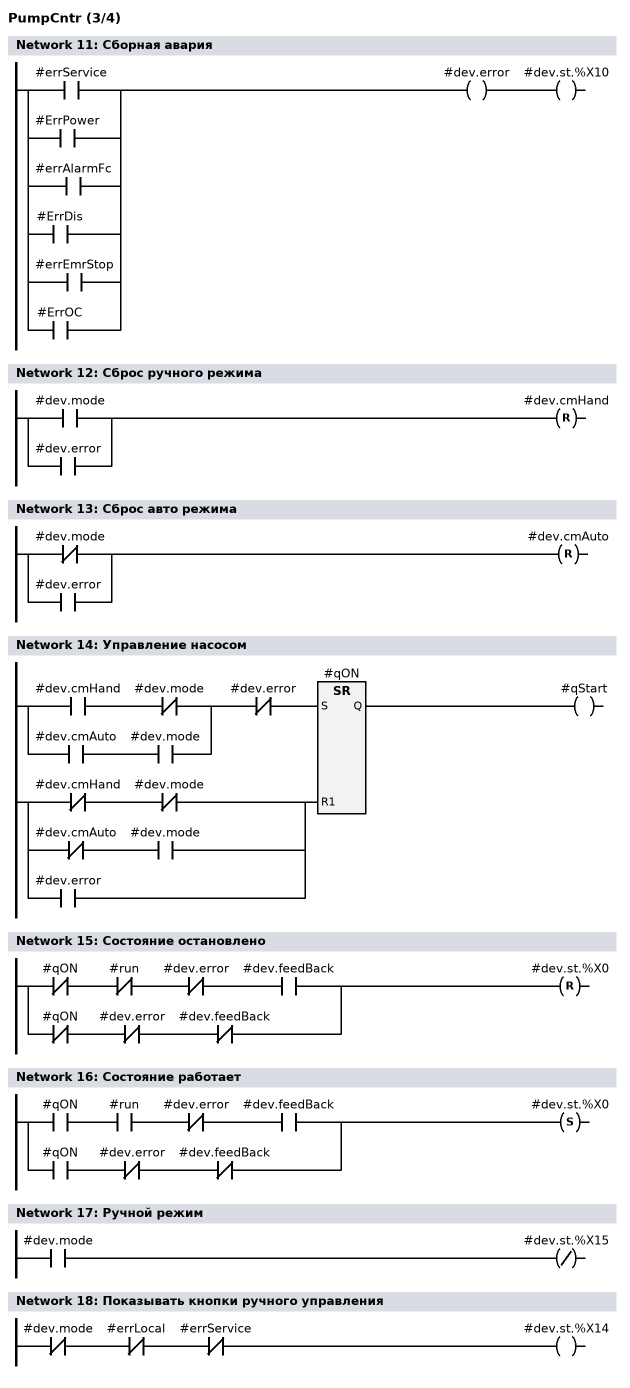
   RUNG wire#powerrail
      Contact( #errService )
      wire#w1
      Coil( #dev.error )
      Coil( #dev.st.%X10 )
   END_RUNG
   RUNG wire#powerrail
      Contact( #ErrPower )
   END_RUNG wire#w1
   RUNG wire#powerrail
      Contact( #errAlarmFc )
   END_RUNG wire#w1
   RUNG wire#powerrail
      Contact( #ErrDis )
   END_RUNG wire#w1
   RUNG wire#powerrail
      Contact( #errEmrStop )
   END_RUNG wire#w1
   RUNG wire#powerrail
      Contact( #ErrOC )
   END_RUNG wire#w1
   // the same network as SCL:
   #dev.error := #errService OR #ErrPower OR #errAlarmFc OR #ErrDis OR #errEmrStop OR #ErrOC;
   #dev.st.%X10 := #dev.error;
END_REGION

REGION Network 12: Сброс ручного режима
   RUNG wire#powerrail
      Contact( #dev.mode )
      wire#w1
      R_Coil( #dev.cmHand )
   END_RUNG
   RUNG wire#powerrail
      Contact( #dev.error )
   END_RUNG wire#w1
   // the same network as SCL:
   IF #dev.mode OR #dev.error THEN #dev.cmHand := FALSE; END_IF;
END_REGION

REGION Network 13: Сброс авто режима
   RUNG wire#powerrail
      I_Contact( #dev.mode )
      wire#w1
      R_Coil( #dev.cmAuto )
   END_RUNG
   RUNG wire#powerrail
      Contact( #dev.error )
   END_RUNG wire#w1
   // the same network as SCL:
   IF NOT #dev.mode OR #dev.error THEN #dev.cmAuto := FALSE; END_IF;
END_REGION

REGION Network 14: Управление насосом
   RUNG wire#powerrail
      Contact( #dev.cmHand )
      I_Contact( #dev.mode )
      wire#w1
      I_Contact( #dev.error )
      S_SR(operand := #qON, r1 := wire#w2)
      Coil( #qStart )
   END_RUNG
   RUNG wire#powerrail
      Contact( #dev.cmAuto )
      Contact( #dev.mode )
   END_RUNG wire#w1
   RUNG wire#powerrail
      I_Contact( #dev.cmHand )
      I_Contact( #dev.mode )
   END_RUNG wire#w2
   RUNG wire#powerrail
      I_Contact( #dev.cmAuto )
      Contact( #dev.mode )
   END_RUNG wire#w2
   RUNG wire#powerrail
      Contact( #dev.error )
   END_RUNG wire#w2
   // the same network as SCL:
   IF ((#dev.cmHand AND NOT #dev.mode) OR (#dev.cmAuto AND #dev.mode)) AND NOT #dev.error THEN
       #qON := TRUE;   // SR flip-flop
   END_IF;
   IF (NOT #dev.cmHand AND NOT #dev.mode) OR (NOT #dev.cmAuto AND #dev.mode) OR #dev.error THEN
       #qON := FALSE;
   END_IF;
   #qStart := #qON;
END_REGION

REGION Network 15: Состояние остановлено
   RUNG wire#powerrail
      I_Contact( #qON )
      I_Contact( #run )
      I_Contact( #dev.error )
      Contact( #dev.feedBack )
      wire#w1
      R_Coil( #dev.st.%X0 )
   END_RUNG
   RUNG wire#powerrail
      I_Contact( #qON )
      I_Contact( #dev.error )
      I_Contact( #dev.feedBack )
   END_RUNG wire#w1
   // the same network as SCL:
   IF (NOT #qON AND NOT #run AND NOT #dev.error AND #dev.feedBack) OR (NOT #qON AND NOT #dev.error AND NOT #dev.feedBack) THEN
       #dev.st.%X0 := FALSE;
   END_IF;
END_REGION

REGION Network 16: Состояние работает
   RUNG wire#powerrail
      Contact( #qON )
      Contact( #run )
      I_Contact( #dev.error )
      Contact( #dev.feedBack )
      wire#w1
      S_Coil( #dev.st.%X0 )
   END_RUNG
   RUNG wire#powerrail
      Contact( #qON )
      I_Contact( #dev.error )
      I_Contact( #dev.feedBack )
   END_RUNG wire#w1
   // the same network as SCL:
   IF (#qON AND #run AND NOT #dev.error AND #dev.feedBack) OR (#qON AND NOT #dev.error AND NOT #dev.feedBack) THEN
       #dev.st.%X0 := TRUE;
   END_IF;
END_REGION

REGION Network 17: Ручной режим
   RUNG wire#powerrail
      Contact( #dev.mode )
      I_Coil( #dev.st.%X15 )
   END_RUNG
   // the same network as SCL:
   #dev.st.%X15 := NOT #dev.mode;
END_REGION

REGION Network 18: Показывать кнопки ручного управления
   RUNG wire#powerrail
      I_Contact( #dev.mode )
      I_Contact( #errLocal )
      I_Contact( #errService )
      Coil( #dev.st.%X14 )
   END_RUNG
   // the same network as SCL:
   #dev.st.%X14 := NOT #dev.mode AND NOT #errLocal AND NOT #errService;
END_REGION

REGION Network 19: Программный выход запуска насоса
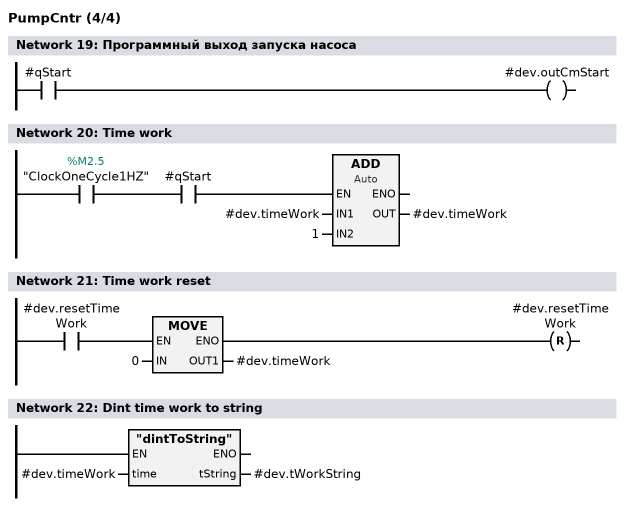
   RUNG wire#powerrail
      Contact( #qStart )
      Coil( #dev.outCmStart )
   END_RUNG
   // the same network as SCL:
   #dev.outCmStart := #qStart;
END_REGION

REGION Network 20: Time work
   RUNG wire#powerrail
      Contact( "ClockOneCycle1HZ" )
      Contact( #qStart )
      Add(in1 := #dev.timeWork, in2 := 1, out => #dev.timeWork)
   END_RUNG
   // the same network as SCL:
   IF "ClockOneCycle1HZ" AND #qStart THEN #dev.timeWork := #dev.timeWork + 1; END_IF;
END_REGION

REGION Network 21: Time work reset
   RUNG wire#powerrail
      Contact( #dev.resetTimeWork )
      Move(in := 0, out1 => #dev.timeWork)
      R_Coil( #dev.resetTimeWork )
   END_RUNG
   // the same network as SCL:
   IF #dev.resetTimeWork THEN
       #dev.timeWork := 0;
       #dev.resetTimeWork := FALSE;
   END_IF;
END_REGION

REGION Network 22: Dint time work to string
   RUNG wire#powerrail
      "dintToString"("time" := #dev.timeWork, tString => #dev.tWorkString)
   END_RUNG
   // the same network as SCL:
   "dintToString"("time" := #dev.timeWork, tString => #dev.tWorkString);
END_REGION
END_FUNCTION_BLOCK

FUNCTION_BLOCK "PumpAckAlarm"   // FB38, LAD
{ S7_Optimized_Access := 'TRUE' }
VERSION : 0.1
// stored: AutoNumber true, IsIECCheckEnabled false, IsRetainMemResEnabled false, MemoryReserve 100, SetENOAutomatically false, UDAEnableTagReadback false
   VAR_INPUT
      ack : Bool;
      power : Bool;
      alarmFC : Bool;
      emrStop : Bool;   // Авариный стоп 0-авария, 1-ок
      local : Bool;   // 1-местный режим
      tmrOpening_Q : Bool;
      tmrClosing_Q : Bool;
   END_VAR
   VAR_IN_OUT
      dev : "Pump";
      errService : Bool;
      ErrPower : Bool;   // Признак аварии питания
      errAlarmFc : Bool;
      ErrDis : Bool;   // Признак внешней блокировки
      errEmrStop : Bool;
      errLocal : Bool;
      errStart : Bool;
      errStop : Bool;
   END_VAR
   VAR
      InstService { S7_SetPoint := 'True'} : "DevAckSingleAlarm";
      InstPower { S7_SetPoint := 'True'} : "DevAckSingleAlarm";
      InstFc { S7_SetPoint := 'True'} : "DevAckSingleAlarm";
      InstDis { S7_SetPoint := 'True'} : "DevBlockAckSingleAlarm";
      InstEmrStop { S7_SetPoint := 'True'} : "DevAckSingleAlarm";
      InstLocal { S7_SetPoint := 'True'} : "DevAckSingleAlarm";
      InstStart { S7_SetPoint := 'True'} : "DevAckSingleAlarm";
      InstStop { S7_SetPoint := 'True'} : "DevAckSingleAlarm";
   END_VAR
BEGIN

REGION Network 1: Сервисный режим - нужно квитирование ACK
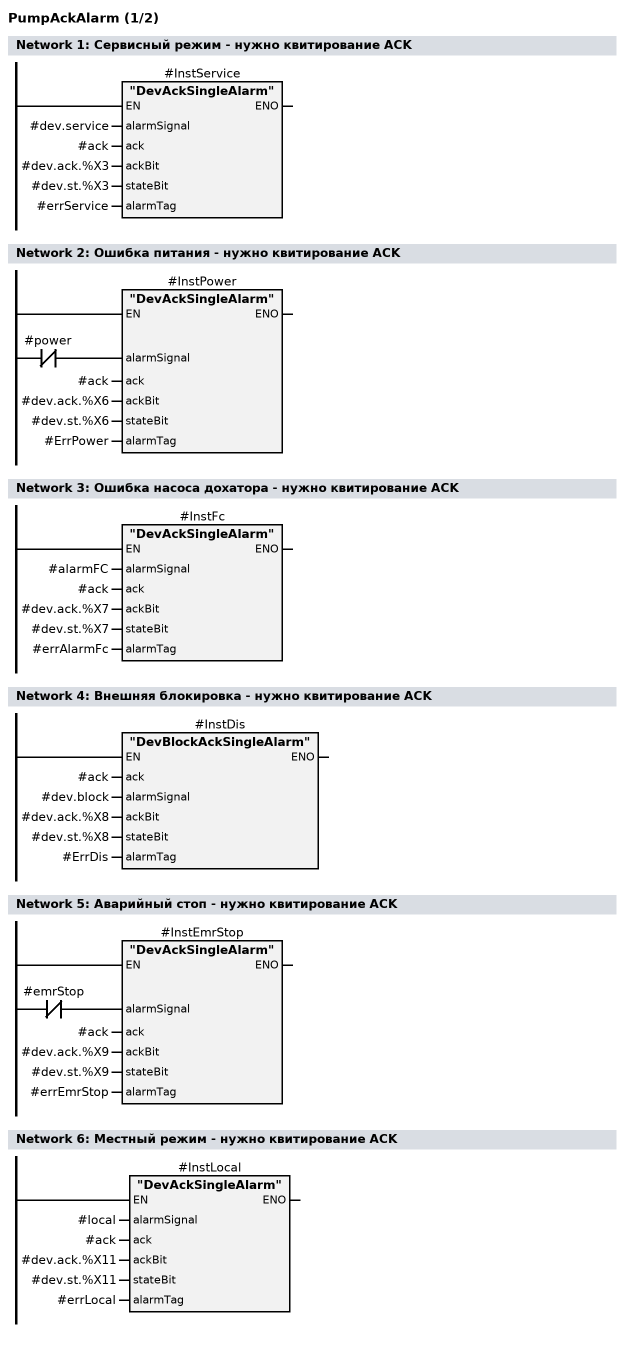
   RUNG wire#powerrail
      #InstService(alarmSignal := #dev.service, ack := #ack, ackBit := #dev.ack.%X3, stateBit := #dev.st.%X3, alarmTag := #errService)
   END_RUNG
   // the same network as SCL:
   #InstService(alarmSignal := #dev.service,   // "DevAckSingleAlarm"
                ack := #ack,
                ackBit := #dev.ack.%X3,
                stateBit := #dev.st.%X3,
                alarmTag := #errService);
END_REGION

REGION Network 2: Ошибка питания - нужно квитирование ACK
   RUNG wire#powerrail
      #InstPower(alarmSignal := wire#w1, ack := #ack, ackBit := #dev.ack.%X6, stateBit := #dev.st.%X6, alarmTag := #ErrPower)
   END_RUNG
   RUNG wire#powerrail
      I_Contact( #power )
   END_RUNG wire#w1
   // the same network as SCL:
   #InstPower(alarmSignal := NOT #power,   // "DevAckSingleAlarm"
              ack := #ack,
              ackBit := #dev.ack.%X6,
              stateBit := #dev.st.%X6,
              alarmTag := #ErrPower);
END_REGION

REGION Network 3: Ошибка насоса дохатора - нужно квитирование ACK
   RUNG wire#powerrail
      #InstFc(alarmSignal := #alarmFC, ack := #ack, ackBit := #dev.ack.%X7, stateBit := #dev.st.%X7, alarmTag := #errAlarmFc)
   END_RUNG
   // the same network as SCL:
   #InstFc(alarmSignal := #alarmFC,   // "DevAckSingleAlarm"
           ack := #ack,
           ackBit := #dev.ack.%X7,
           stateBit := #dev.st.%X7,
           alarmTag := #errAlarmFc);
END_REGION

REGION Network 4: Внешняя блокировка - нужно квитирование ACK
   RUNG wire#powerrail
      #InstDis(ack := #ack, alarmSignal := #dev.block, ackBit := #dev.ack.%X8, stateBit := #dev.st.%X8, alarmTag := #ErrDis)
   END_RUNG
   // the same network as SCL:
   #InstDis(ack := #ack,   // "DevBlockAckSingleAlarm"
            alarmSignal := #dev.block,
            ackBit := #dev.ack.%X8,
            stateBit := #dev.st.%X8,
            alarmTag := #ErrDis);
END_REGION

REGION Network 5: Аварийный стоп - нужно квитирование ACK
   RUNG wire#powerrail
      #InstEmrStop(alarmSignal := wire#w1, ack := #ack, ackBit := #dev.ack.%X9, stateBit := #dev.st.%X9, alarmTag := #errEmrStop)
   END_RUNG
   RUNG wire#powerrail
      I_Contact( #emrStop )
   END_RUNG wire#w1
   // the same network as SCL:
   #InstEmrStop(alarmSignal := NOT #emrStop,   // "DevAckSingleAlarm"
                ack := #ack,
                ackBit := #dev.ack.%X9,
                stateBit := #dev.st.%X9,
                alarmTag := #errEmrStop);
END_REGION

REGION Network 6: Местный режим - нужно квитирование ACK
   RUNG wire#powerrail
      #InstLocal(alarmSignal := #local, ack := #ack, ackBit := #dev.ack.%X11, stateBit := #dev.st.%X11, alarmTag := #errLocal)
   END_RUNG
   // the same network as SCL:
   #InstLocal(alarmSignal := #local,   // "DevAckSingleAlarm"
              ack := #ack,
              ackBit := #dev.ack.%X11,
              stateBit := #dev.st.%X11,
              alarmTag := #errLocal);
END_REGION

REGION Network 7: Состояние ошибки запуска ACK
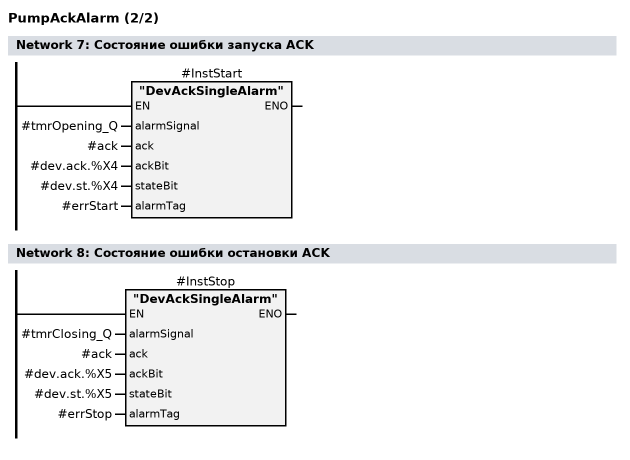
   RUNG wire#powerrail
      #InstStart(alarmSignal := #tmrOpening_Q, ack := #ack, ackBit := #dev.ack.%X4, stateBit := #dev.st.%X4, alarmTag := #errStart)
   END_RUNG
   // the same network as SCL:
   #InstStart(alarmSignal := #tmrOpening_Q,   // "DevAckSingleAlarm"
              ack := #ack,
              ackBit := #dev.ack.%X4,
              stateBit := #dev.st.%X4,
              alarmTag := #errStart);
END_REGION

REGION Network 8: Состояние ошибки остановки ACK
   RUNG wire#powerrail
      #InstStop(alarmSignal := #tmrClosing_Q, ack := #ack, ackBit := #dev.ack.%X5, stateBit := #dev.st.%X5, alarmTag := #errStop)
   END_RUNG
   // the same network as SCL:
   #InstStop(alarmSignal := #tmrClosing_Q,   // "DevAckSingleAlarm"
             ack := #ack,
             ackBit := #dev.ack.%X5,
             stateBit := #dev.st.%X5,
             alarmTag := #errStop);
END_REGION
END_FUNCTION_BLOCK

FUNCTION_BLOCK "DevAckSingleAlarm"   // FB39, LAD
{ S7_Optimized_Access := 'TRUE' }
VERSION : 0.1
// stored: AutoNumber true, IsIECCheckEnabled false, IsRetainMemResEnabled false, MemoryReserve 100, SetENOAutomatically false, UDAEnableTagReadback false
   VAR_INPUT
      alarmSignal : Bool;
      ack : Bool;
   END_VAR
   VAR_IN_OUT
      ackBit : Bool;
      stateBit : Bool;
      alarmTag : Bool;
   END_VAR
   VAR
      ACK_TAG : TON_TIME;
   END_VAR
   VAR CONSTANT
      ACK_DELAY : Time := T#1s;
   END_VAR
BEGIN

REGION Network 1
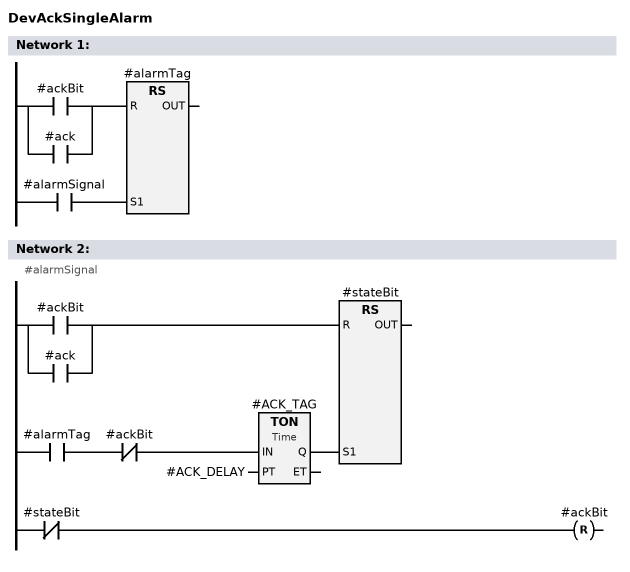
   RUNG wire#powerrail
      Contact( #ackBit )
      wire#w1
      S_RS(operand := #alarmTag, s1 := wire#w2)
   END_RUNG
   RUNG wire#powerrail
      Contact( #ack )
   END_RUNG wire#w1
   RUNG wire#powerrail
      Contact( #alarmSignal )
   END_RUNG wire#w2
   // the same network as SCL:
   IF #ackBit OR #ack THEN
       #alarmTag := FALSE;   // RS flip-flop
   END_IF;
   IF #alarmSignal THEN #alarmTag := TRUE; END_IF;
END_REGION

REGION Network 2
   // #alarmSignal
   RUNG wire#powerrail
      Contact( #ackBit )
      wire#w1
      S_RS(operand := #stateBit, s1 := wire#w2)
   END_RUNG
   RUNG wire#powerrail
      Contact( #ack )
   END_RUNG wire#w1
   RUNG wire#powerrail
      Contact( #alarmTag )
      I_Contact( #ackBit )
      { S7_Templates := "time_type := Time" } #ACK_TAG.TON(pt := #ACK_DELAY, et =>)
   END_RUNG wire#w2
   RUNG wire#powerrail
      I_Contact( #stateBit )
      R_Coil( #ackBit )
   END_RUNG
   // the same network as SCL:
   #ACK_TAG(IN := #alarmTag AND NOT #ackBit, PT := #ACK_DELAY);   // TON
   IF #ackBit OR #ack THEN
       #stateBit := FALSE;   // RS flip-flop
   END_IF;
   IF #ACK_TAG.Q THEN #stateBit := TRUE; END_IF;
   IF NOT #stateBit THEN #ackBit := FALSE; END_IF;
END_REGION
END_FUNCTION_BLOCK

FUNCTION_BLOCK "DevBlockAckSingleAlarm"   // FB55, LAD
{ S7_Optimized_Access := 'TRUE' }
VERSION : 0.1
// stored: AutoNumber true, IsIECCheckEnabled false, IsRetainMemResEnabled false, MemoryReserve 100, SetENOAutomatically false, UDAEnableTagReadback false
   VAR_INPUT
      ack : Bool;
   END_VAR
   VAR_IN_OUT
      alarmSignal : Bool;
      ackBit : Bool;
      stateBit : Bool;
      alarmTag : Bool;
   END_VAR
   VAR
      ACK_TAG : TON_TIME;
   END_VAR
   VAR CONSTANT
      ACK_DELAY : Time := T#2s;
   END_VAR
BEGIN

REGION Network 1
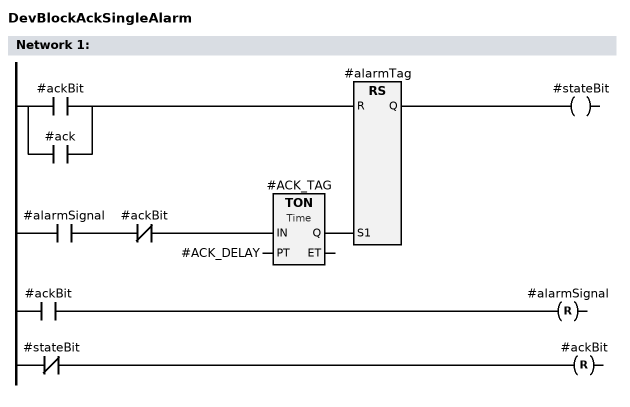
   RUNG wire#powerrail
      Contact( #ackBit )
      wire#w1
      S_RS(operand := #alarmTag, s1 := wire#w2)
      Coil( #stateBit )
   END_RUNG
   RUNG wire#powerrail
      Contact( #ack )
   END_RUNG wire#w1
   RUNG wire#powerrail
      Contact( #alarmSignal )
      I_Contact( #ackBit )
      { S7_Templates := "time_type := Time" } #ACK_TAG.TON(pt := #ACK_DELAY, et =>)
   END_RUNG wire#w2
   RUNG wire#powerrail
      Contact( #ackBit )
      R_Coil( #alarmSignal )
   END_RUNG
   RUNG wire#powerrail
      I_Contact( #stateBit )
      R_Coil( #ackBit )
   END_RUNG
   // the same network as SCL:
   #ACK_TAG(IN := #alarmSignal AND NOT #ackBit, PT := #ACK_DELAY);   // TON
   IF #ackBit OR #ack THEN
       #alarmTag := FALSE;   // RS flip-flop
   END_IF;
   IF #ACK_TAG.Q THEN #alarmTag := TRUE; END_IF;
   #stateBit := #alarmTag;
   IF #ackBit THEN #alarmSignal := FALSE; END_IF;
   IF NOT #stateBit THEN #ackBit := FALSE; END_IF;
END_REGION
END_FUNCTION_BLOCK

FUNCTION_BLOCK "hardwareTimePulse"   // FB12, FBD
{ S7_Optimized_Access := 'FALSE' }
VERSION : 0.1
// stored: AutoNumber false, IsIECCheckEnabled false, SetENOAutomatically false, UDAEnableTagReadback false
   VAR DB_SPECIFIC
      pTrig1HZ : Bool;
      pTrig05Hz : Bool;
      pTrig0625Hz : Bool;
      pTrig1_25HZ : Bool;
      pTrig2HZ : Bool;
      pTrig2_5Hz : Bool;
      pTirg5Hz : Bool;
      pTrig10Hz : Bool;
   END_VAR
   VAR_TEMP   // added for the SCL form of the ladder/FBD networks
      _w1 : Bool;
   END_VAR
BEGIN

REGION Network 1
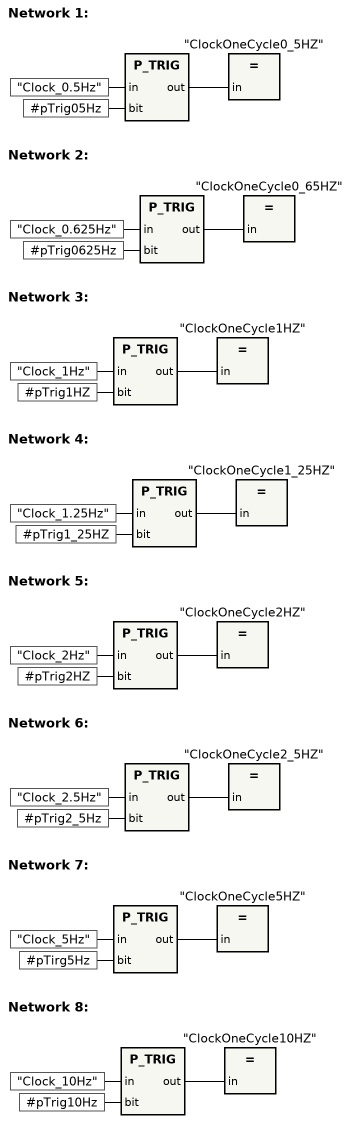
   #_w1 := "Clock_0.5Hz" AND NOT #pTrig05Hz;   // rising edge
   #pTrig05Hz := "Clock_0.5Hz";
   "ClockOneCycle0_5HZ" := #_w1;
END_REGION

REGION Network 2
   #_w1 := "Clock_0.625Hz" AND NOT #pTrig0625Hz;   // rising edge
   #pTrig0625Hz := "Clock_0.625Hz";
   "ClockOneCycle0_65HZ" := #_w1;
END_REGION

REGION Network 3
   #_w1 := "Clock_1Hz" AND NOT #pTrig1HZ;   // rising edge
   #pTrig1HZ := "Clock_1Hz";
   "ClockOneCycle1HZ" := #_w1;
END_REGION

REGION Network 4
   #_w1 := "Clock_1.25Hz" AND NOT #pTrig1_25HZ;   // rising edge
   #pTrig1_25HZ := "Clock_1.25Hz";
   "ClockOneCycle1_25HZ" := #_w1;
END_REGION

REGION Network 5
   #_w1 := "Clock_2Hz" AND NOT #pTrig2HZ;   // rising edge
   #pTrig2HZ := "Clock_2Hz";
   "ClockOneCycle2HZ" := #_w1;
END_REGION

REGION Network 6
   #_w1 := "Clock_2.5Hz" AND NOT #pTrig2_5Hz;   // rising edge
   #pTrig2_5Hz := "Clock_2.5Hz";
   "ClockOneCycle2_5HZ" := #_w1;
END_REGION

REGION Network 7
   #_w1 := "Clock_5Hz" AND NOT #pTirg5Hz;   // rising edge
   #pTirg5Hz := "Clock_5Hz";
   "ClockOneCycle5HZ" := #_w1;
END_REGION

REGION Network 8
   #_w1 := "Clock_10Hz" AND NOT #pTrig10Hz;   // rising edge
   #pTrig10Hz := "Clock_10Hz";
   "ClockOneCycle10HZ" := #_w1;
END_REGION
END_FUNCTION_BLOCK

FUNCTION "levelSelect" : Void
{ S7_Optimized_Access := 'TRUE' }
VERSION : 0.1
   VAR_INPUT 
      sel : Int;   // 0-1+2, 1-1, 2-2
      levelTank1 : Real;
      levelTank2 : Real;
   END_VAR

   VAR_OUTPUT 
      work1 : Bool;   // 0-reserv, 1-work
      work2 : Bool;   // 0-reserv, 1-work
      level : Real;
   END_VAR


BEGIN
	CASE #sel OF
	    0:
	        #work1 := 1;
	        #work2 := 1;
	        #level := (#levelTank1 + #levelTank2) / 2.0;
	    1:
	        #work1 := 1;
	        #work2 := 0;
	        #level := #levelTank1;
	    2:
	        #work1 := 0;
	        #work2 := 1;
	        #level := #levelTank2;
	    ELSE  // Statement section ELSE
	        #work1 := 1;
	        #work2 := 1;
	        #level := 351.0;
	END_CASE;
	
END_FUNCTION

FUNCTION_BLOCK "AllDigital"   // FB5, FBD
{ S7_Optimized_Access := 'TRUE' }
VERSION : 0.1
// stored: AutoNumber true, IsIECCheckEnabled false, IsRetainMemResEnabled false, MemoryReserve 100, SetENOAutomatically false, UDAEnableTagReadback false
   VAR
      FL501 { S7_SetPoint := 'True'} : "DigitalSensorCntrl";
      FL901 { S7_SetPoint := 'True'} : "DigitalSensorCntrl";
      FL1301 { S7_SetPoint := 'True'} : "DigitalSensorCntrl";
      PS901 { S7_SetPoint := 'True'} : "DigitalSensorCntrl";
      PS902 { S7_SetPoint := 'True'} : "DigitalSensorCntrl";
      PS1301 { S7_SetPoint := 'True'} : "DigitalSensorCntrl";
      PS1302 { S7_SetPoint := 'True'} : "DigitalSensorCntrl";
   END_VAR
BEGIN

REGION Network 1: 1-включить детектирование аварии
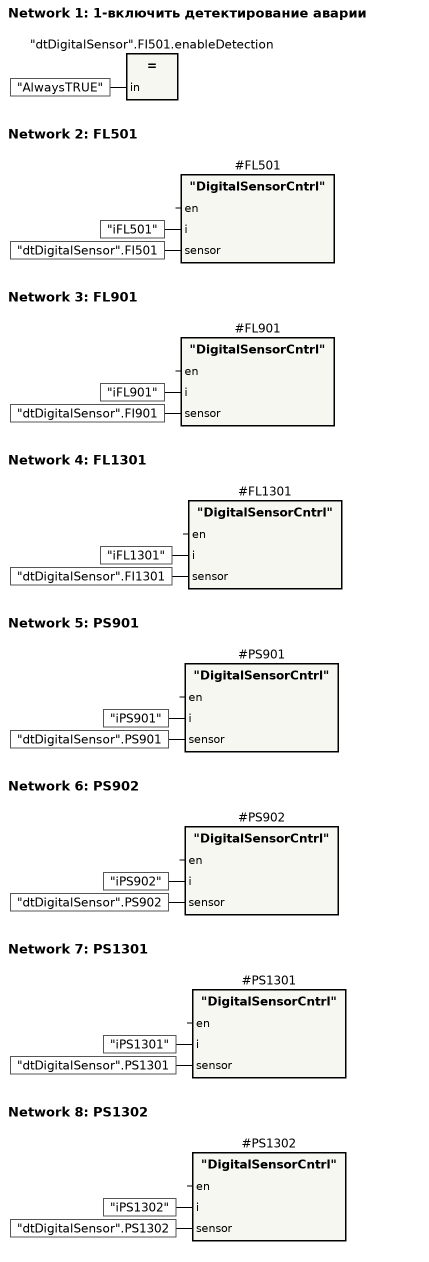
   "dtDigitalSensor".FI501.enableDetection := "AlwaysTRUE";
END_REGION

REGION Network 2: FL501
   #FL501(i := "iFL501", sensor := "dtDigitalSensor".FI501);   // "DigitalSensorCntrl"
END_REGION

REGION Network 3: FL901
   #FL901(i := "iFL901", sensor := "dtDigitalSensor".FI901);   // "DigitalSensorCntrl"
END_REGION

REGION Network 4: FL1301
   #FL1301(i := "iFL1301", sensor := "dtDigitalSensor".FI1301);   // "DigitalSensorCntrl"
END_REGION

REGION Network 5: PS901
   #PS901(i := "iPS901", sensor := "dtDigitalSensor".PS901);   // "DigitalSensorCntrl"
END_REGION

REGION Network 6: PS902
   #PS902(i := "iPS902", sensor := "dtDigitalSensor".PS902);   // "DigitalSensorCntrl"
END_REGION

REGION Network 7: PS1301
   #PS1301(i := "iPS1301", sensor := "dtDigitalSensor".PS1301);   // "DigitalSensorCntrl"
END_REGION

REGION Network 8: PS1302
   #PS1302(i := "iPS1302", sensor := "dtDigitalSensor".PS1302);   // "DigitalSensorCntrl"
END_REGION
END_FUNCTION_BLOCK

FUNCTION_BLOCK "DigitalSensorCntrl"   // FB80, FBD
{ S7_Optimized_Access := 'TRUE' }
VERSION : 0.1
// выход 1-авария
// в режиме авто, прямой вход - 0-авария, с инверсией - 1-авария
// в ручном режиме включение авария -
// stored: AutoNumber false, IsIECCheckEnabled false, IsRetainMemResEnabled false, MemoryReserve 100, SetENOAutomatically false, UDAEnableTagReadback false
   VAR_INPUT
      i : Bool;
   END_VAR
   VAR_IN_OUT
      sensor : "digitalSensor";
   END_VAR
BEGIN

REGION Network 1: Промежуточное состояние без задержки
   // 1-alarm
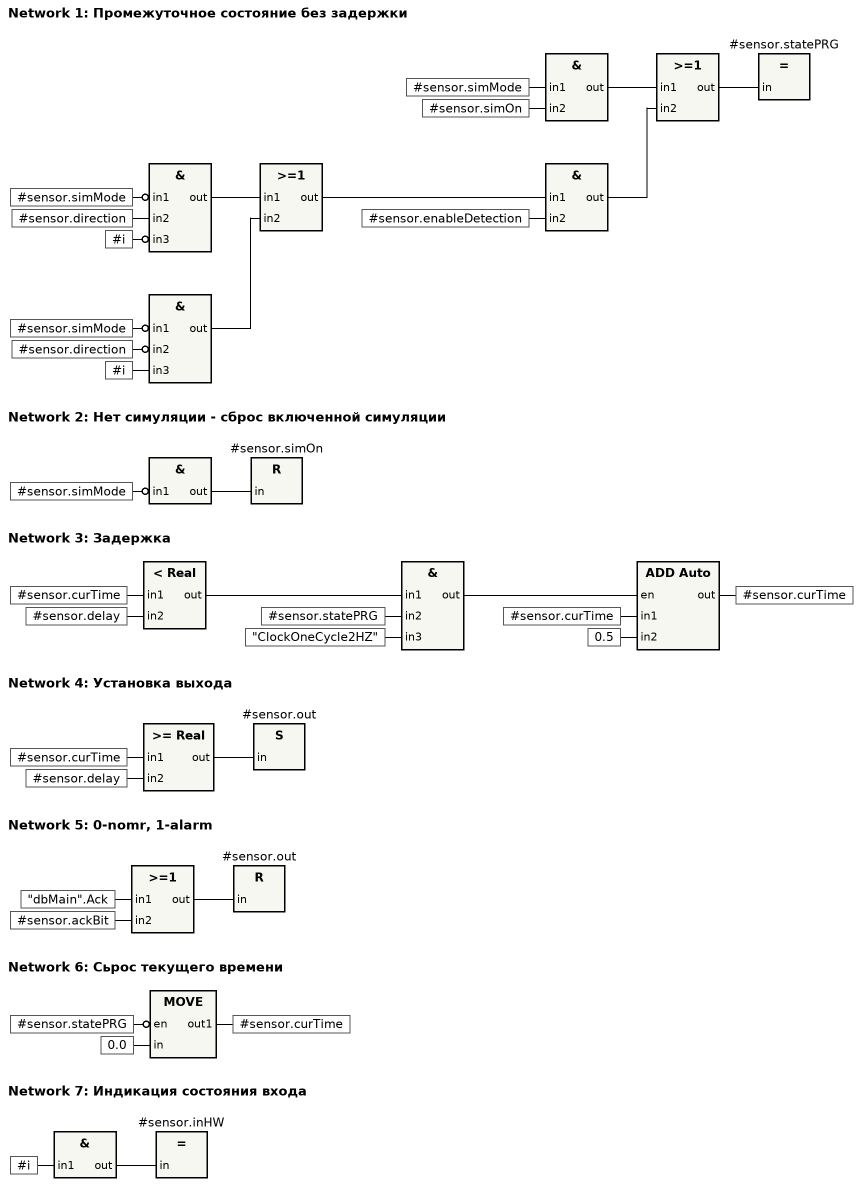
   #sensor.statePRG := (#sensor.simMode AND #sensor.simOn) OR (((NOT #sensor.simMode AND #sensor.direction AND NOT #i) OR (NOT #sensor.simMode AND NOT #sensor.direction AND #i)) AND #sensor.enableDetection);
END_REGION

REGION Network 2: Нет симуляции - сброс включенной симуляции
   IF NOT #sensor.simMode THEN #sensor.simOn := FALSE; END_IF;
END_REGION

REGION Network 3: Задержка
   IF (#sensor.curTime < #sensor.delay) AND #sensor.statePRG AND "ClockOneCycle2HZ" THEN
       #sensor.curTime := #sensor.curTime + 0.5;
   END_IF;
END_REGION

REGION Network 4: Установка выхода
   IF #sensor.curTime >= #sensor.delay THEN #sensor.out := TRUE; END_IF;
END_REGION

REGION Network 5: 0-nomr, 1-alarm
   IF "dbMain".Ack OR #sensor.ackBit THEN #sensor.out := FALSE; END_IF;
END_REGION

REGION Network 6: Сьрос текущего времени
   IF NOT #sensor.statePRG THEN #sensor.curTime := 0.0; END_IF;
END_REGION

REGION Network 7: Индикация состояния входа
   #sensor.inHW := #i;
END_REGION
END_FUNCTION_BLOCK

FUNCTION_BLOCK "AllFlowCounter"
{ S7_Optimized_Access := 'TRUE' }
VERSION : 0.1
   VAR 
      prewHour : USInt;
      prewDay : USInt;
      FM201 : "VolumeCounter";
      FM501 : "VolumeCounter";
      FM502 : "VolumeCounter";
      FM901 : "VolumeCounter";
      FM902 : "VolumeCounter";
      FM1201 : "VolumeCounter";
      FM1301 : "VolumeCounter";
      FM1302 : "VolumeCounter";
      FM1701 : "VolumeCounter";
      FM1801 : "VolumeCounter";
   END_VAR

   VAR_TEMP 
      tRetInt : Int;
      tCurTime {InstructionName := 'DTL'; LibVersion := '1.0'} : DTL;
      tNextHour : Bool;
      tNextDay : Bool;
   END_VAR


BEGIN
	#tRetInt := RD_LOC_T(#tCurTime);
	IF #tCurTime.HOUR <> #prewHour THEN
	    #prewHour := #tCurTime.HOUR;
	    #tNextHour := TRUE;
	END_IF;
	IF #tCurTime.DAY <> #prewDay THEN
	    #prewDay := #tCurTime.DAY;
	    #tNextDay := TRUE;
	END_IF;
	#FM201(puls:="iFM201",
	       nextHour:=#tNextHour,
	       nextDay:=#tNextDay,
	       data:="dbVolumeCounters".FM201);
	#FM501(puls := "iFM501",
	       nextHour := #tNextHour,
	       nextDay := #tNextDay,
	       data := "dbVolumeCounters".FM501);
	#FM502(puls := "iFM502",
	       nextHour := #tNextHour,
	       nextDay := #tNextDay,
	       data := "dbVolumeCounters".FM502);
	#FM901(puls := "iFM901",
	       nextHour := #tNextHour,
	       nextDay := #tNextDay,
	       data := "dbVolumeCounters".FM901);
	#FM902(puls := "iFM902",
	       nextHour := #tNextHour,
	       nextDay := #tNextDay,
	       data := "dbVolumeCounters".FM902);
	#FM1201(puls := "iFM1201",
	        nextHour := #tNextHour,
	        nextDay := #tNextDay,
	        data := "dbVolumeCounters".FM1201);
	#FM1301(puls := "iFM1301",
	        nextHour := #tNextHour,
	        nextDay := #tNextDay,
	        data := "dbVolumeCounters".FM1301);
	#FM1302(puls := "iFM1302",
	        nextHour := #tNextHour,
	        nextDay := #tNextDay,
	        data := "dbVolumeCounters".FM1302);
	#FM1701(puls := "iFM1701",
	        nextHour := #tNextHour,
	        nextDay := #tNextDay,
	        data := "dbVolumeCounters".FM1701);
	#FM1801(puls := "iFM1801",
	        nextHour := #tNextHour,
	        nextDay := #tNextDay,
	        data := "dbVolumeCounters".FM1801);
END_FUNCTION_BLOCK

FUNCTION_BLOCK "VolumeCounter"   // FB65, FBD
{ S7_Optimized_Access := 'TRUE' }
VERSION : 0.1
// stored: AutoNumber true, IsIECCheckEnabled false, IsRetainMemResEnabled false, MemoryReserve 100, SetENOAutomatically false, UDAEnableTagReadback false
   VAR_INPUT
      puls : Bool;
      nextHour : Bool;
      nextDay : Bool;
   END_VAR
   VAR_IN_OUT
      data : "FREQ_COUNTER";
   END_VAR
   VAR
      litrs : UInt;
      pTrig : Bool;
   END_VAR
   VAR CONSTANT
      FB_CALL_TIME : Real := 0.1;
   END_VAR
   VAR_TEMP   // added for the SCL form of the ladder/FBD networks
      _w1 : Bool;
   END_VAR
BEGIN

REGION Network 1: Add to counter
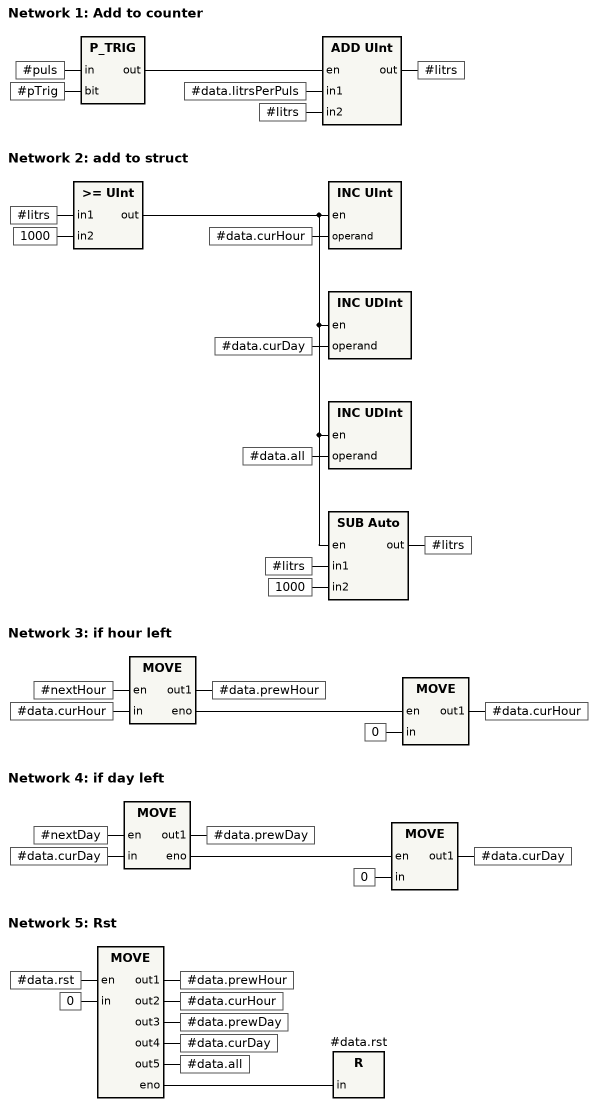
   #_w1 := #puls AND NOT #pTrig;   // rising edge
   #pTrig := #puls;
   IF #_w1 THEN #litrs := #data.litrsPerPuls + #litrs; END_IF;
END_REGION

REGION Network 2: add to struct
   IF #litrs >= 1000 THEN
       #data.curHour := #data.curHour + 1;
       #data.curDay := #data.curDay + 1;
       #data.all := #data.all + 1;
       #litrs := #litrs - 1000;
   END_IF;
END_REGION

REGION Network 3: if hour left
   IF #nextHour THEN
       #data.prewHour := #data.curHour;
       #data.curHour := 0;
   END_IF;
END_REGION

REGION Network 4: if day left
   IF #nextDay THEN
       #data.prewDay := #data.curDay;
       #data.curDay := 0;
   END_IF;
END_REGION

REGION Network 5: Rst
   IF #data.rst THEN
       #data.prewHour := 0;
       #data.curHour := 0;
       #data.prewDay := 0;
       #data.curDay := 0;
       #data.all := 0;
       #data.rst := FALSE;
   END_IF;
END_REGION
END_FUNCTION_BLOCK

ORGANIZATION_BLOCK "Cyclic interrupt"   // OB30, LAD, CyclicInterrupt
{ S7_Optimized_Access := 'TRUE' }
VERSION : 0.1
// stored: AutoNumber true, IsIECCheckEnabled false, SetENOAutomatically false
   VAR_INPUT
      Initial_Call : Bool;   // Initial call of this OB
      Event_Count : Int;   // Events discarded
   END_VAR
BEGIN

REGION Network 1: Plc analogs
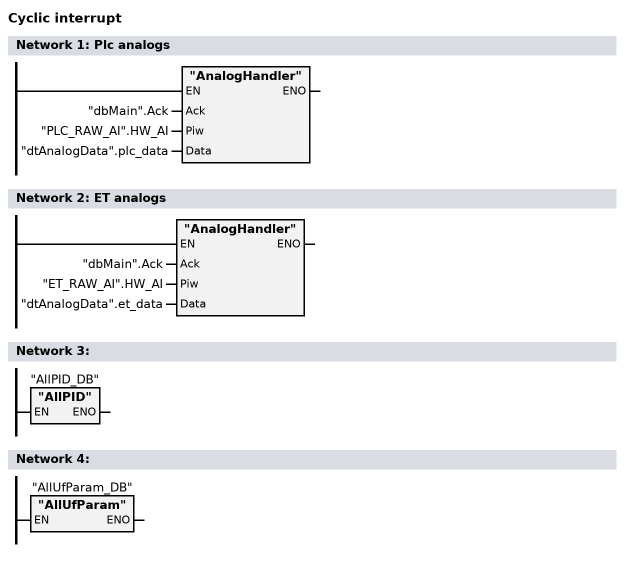
   RUNG wire#powerrail
      "AnalogHandler"(Ack := "dbMain".Ack, Piw := "PLC_RAW_AI".HW_AI, Data := "dtAnalogData".plc_data)
   END_RUNG
   // the same network as SCL:
   "AnalogHandler"(Ack := "dbMain".Ack, Piw := "PLC_RAW_AI".HW_AI, Data := "dtAnalogData".plc_data);
END_REGION

REGION Network 2: ET analogs
   RUNG wire#powerrail
      "AnalogHandler"(Ack := "dbMain".Ack, Piw := "ET_RAW_AI".HW_AI, Data := "dtAnalogData".et_data)
   END_RUNG
   // the same network as SCL:
   "AnalogHandler"(Ack := "dbMain".Ack, Piw := "ET_RAW_AI".HW_AI, Data := "dtAnalogData".et_data);
END_REGION

REGION Network 3
   RUNG wire#powerrail
      "AllPID_DB"()
   END_RUNG
   // the same network as SCL:
   "AllPID_DB"();   // "AllPID"
END_REGION

REGION Network 4
   RUNG wire#powerrail
      "AllUfParam_DB"()
   END_RUNG
   // the same network as SCL:
   "AllUfParam_DB"();   // "AllUfParam"
END_REGION
END_ORGANIZATION_BLOCK

FUNCTION "AnalogHandler" : Void   // FC1, FBD
{ S7_Optimized_Access := 'TRUE' }
VERSION : 0.1
// stored: AutoNumber true, IsIECCheckEnabled false, SetENOAutomatically false, UDAEnableTagReadback false
   VAR_INPUT
      Ack : Bool;
      Piw : Array[*] of Int;
   END_VAR
   VAR_IN_OUT
      Data : Array[*] of "Ai";
   END_VAR
   VAR_TEMP
      tLb : Int;
      tUb : Int;
      i : Int;
   END_VAR
   VAR CONSTANT
      ERROR : Word := 16#01;
      BAD_PARAMETRS : Word := 16#02;
      HARDWARE_FAULT : Word := 16#04;
      SIMULATION : Word := 16#08;
      EMERGENCY_MIN : Word := 16#10;
      WARNING_MIN : Word := 16#20;
      WARNING_MAX : Word := 16#40;
      EMERGENCY_MAX : Word := 16#80;
   END_VAR
BEGIN

REGION Network 1 (SCL)
   #tLb := DINT_TO_INT(LOWER_BOUND(ARR := #Data, DIM := 1));
   #tUb := DINT_TO_INT(UPPER_BOUND(ARR := #Data, DIM := 1));

   FOR #i := #tLb TO #tUb DO
       #Data[#i].Par_code := #Piw[#i];
       #Data[#i].Par_mA := 4.0 + 16.0 * INT_TO_REAL(#Data[#i].Par_code) / 27648.0;

       IF #Data[#i].SimEnable THEN
           #Data[#i].badParam := #Data[#i].wireBreak := #Data[#i].overFlow := FALSE;
       ELSE
           #Data[#i].badParam := #Data[#i].rngUpLm < #Data[#i].rngLwLm;
           #Data[#i].wireBreak := #Data[#i].Par_code < -4866;//1.185 mA
           #Data[#i].overFlow := #Data[#i].Par_code > 32511; //22.81 mA
       END_IF;
       #Data[#i].Err :=
       #Data[#i].badParam OR
       #Data[#i].wireBreak OR
       #Data[#i].overFlow;

       IF #Data[#i].SimEnable THEN
           #Data[#i].Par := #Data[#i].SimValue;
       ELSE
           IF NOT #Data[#i].Err THEN
               #Data[#i].Par := #Data[#i].rngLwLm + INT_TO_REAL(#Data[#i].Par_code) * (#Data[#i].rngUpLm - #Data[#i].rngLwLm) / 27648.0;
               IF #Data[#i].disableParLessZero AND #Data[#i].Par < 0.0 THEN
                   #Data[#i].Par := 0.0;
               END_IF;
           ELSE
               #Data[#i].Par := 0;
           END_IF;
       END_IF;
       //Flags
       IF #Data[#i].Err THEN
           "setFlags"(enCondition := FALSE,
                      condition := #Data[#i].Par < #Data[#i].emrMin,
                      setTimerVal := #Data[#i].emrMinTime,
                      curFlag := #Data[#i].curEmMin,
                      mainFlag := #Data[#i].emMin,
                      timerVal := #Data[#i].curTimeEmrMin);
           "setFlags"(enCondition := FALSE,
                      condition := #Data[#i].Par > #Data[#i].emrMax,
                      setTimerVal := #Data[#i].emrMaxTime,
                      curFlag := #Data[#i].curEmMax,
                      mainFlag := #Data[#i].emMax,
                      timerVal := #Data[#i].curTimeEmrMax);
           "setFlags"(enCondition := FALSE,
                      condition := #Data[#i].Par < #Data[#i].wrnMin,
                      setTimerVal := #Data[#i].wrnMinTime,
                      curFlag := #Data[#i].curWnMin,
                      mainFlag := #Data[#i].wnMin,
                      timerVal := #Data[#i].curTimeWrnMin);
           "setFlags"(enCondition := FALSE,
                      condition := #Data[#i].Par > #Data[#i].wrnMax,
                      setTimerVal := #Data[#i].wrnMaxTime,
                      curFlag := #Data[#i].curWnMax,
                      mainFlag := #Data[#i].wnMax,
                      timerVal := #Data[#i].curTimeWrnMax);
           ELSE
           "setFlags"(enCondition:=#Data[#i].emMin_En,
                      condition:=#Data[#i].Par < #Data[#i].emrMin,
                      setTimerVal:=#Data[#i].emrMinTime,
                      curFlag:=#Data[#i].curEmMin,
                      mainFlag:=#Data[#i].emMin,
                      timerVal:=#Data[#i].curTimeEmrMin);
           "setFlags"(enCondition := #Data[#i].emMax_En,
                      condition := #Data[#i].Par > #Data[#i].emrMax,
                      setTimerVal := #Data[#i].emrMaxTime,
                      curFlag := #Data[#i].curEmMax,
                      mainFlag := #Data[#i].emMax,
                      timerVal := #Data[#i].curTimeEmrMax);
           "setFlags"(enCondition := #Data[#i].wrnMin_En,
                      condition := #Data[#i].Par < #Data[#i].wrnMin,
                      setTimerVal := #Data[#i].wrnMinTime,
                      curFlag := #Data[#i].curWnMin,
                      mainFlag := #Data[#i].wnMin,
                      timerVal := #Data[#i].curTimeWrnMin);
           "setFlags"(enCondition := #Data[#i].wrnMax_En,
                      condition := #Data[#i].Par > #Data[#i].wrnMax,
                      setTimerVal := #Data[#i].wrnMaxTime,
                      curFlag := #Data[#i].curWnMax,
                      mainFlag := #Data[#i].wnMax,
                      timerVal := #Data[#i].curTimeWrnMax);
       END_IF;
       //Ack
   //    #Data[#i].ackAll := #Ack;
       IF #Data[#i].modeAck THEN
           IF #Data[#i].ackAll THEN
               #Data[#i].emMin := #Data[#i].emMax := #Data[#i].wnMin := #Data[#i].wnMax := FALSE;
               #Data[#i].curTimeEmrMin := #Data[#i].curTimeEmrMax := #Data[#i].curTimeWrnMin := #Data[#i].curTimeWrnMax := 0;
           END_IF;
           IF (#Data[#i].ack AND 16#10) > 0 THEN
               #Data[#i].emMin := FALSE;
               #Data[#i].curTimeEmrMin := 0;
               #Data[#i].ack := #Data[#i].ack AND NOT(DWORD_TO_BYTE(#EMERGENCY_MIN));
           END_IF;
           IF (#Data[#i].ack AND 16#80) > 0 THEN
               #Data[#i].emMax := FALSE;
               #Data[#i].curTimeEmrMax := 0;
               #Data[#i].ack := #Data[#i].ack AND NOT(DWORD_TO_BYTE(#EMERGENCY_MAX));
           END_IF;
       ELSE
           IF NOT #Data[#i].curEmMin THEN
               #Data[#i].emMin := FALSE;
           END_IF;
           IF NOT #Data[#i].curEmMax THEN
               #Data[#i].emMax := FALSE;
           END_IF;
       END_IF;
       //Rst warning flags after normalization value
       IF NOT #Data[#i].curWnMin THEN
           #Data[#i].wnMin := FALSE;
       END_IF;
       IF NOT #Data[#i].curWnMax THEN
           #Data[#i].wnMax := FALSE;
       END_IF;
       //States:
       "setState"(condition:= NOT #Data[#i].Err,
                  hexVal:=#ERROR,
                  state:=#Data[#i].State);
       "setState"(condition := #Data[#i].badParam,
                  hexVal := #BAD_PARAMETRS,
                  state := #Data[#i].State);
       "setState"(condition := #Data[#i].wireBreak OR #Data[#i].overFlow,
                  hexVal := #HARDWARE_FAULT,
                  state := #Data[#i].State);
       "setState"(condition := #Data[#i].SimEnable,
                  hexVal := #SIMULATION,
                  state := #Data[#i].State);
       "setState"(condition := #Data[#i].emMin,
                  hexVal := #EMERGENCY_MIN,
                  state := #Data[#i].State);
       "setState"(condition := #Data[#i].wnMin,
                  hexVal := #WARNING_MIN,
                  state := #Data[#i].State);
       "setState"(condition := #Data[#i].wnMax,
                  hexVal := #WARNING_MAX,
                  state := #Data[#i].State);
       "setState"(condition := #Data[#i].emMax,
                  hexVal := #EMERGENCY_MAX,
                  state := #Data[#i].State);
   END_FOR;
END_REGION
END_FUNCTION

FUNCTION_BLOCK "AllPID"   // FB3, FBD
{ S7_Optimized_Access := 'TRUE' }
VERSION : 0.1
// stored: AutoNumber true, IsIECCheckEnabled false, IsRetainMemResEnabled false, MemoryReserve 100, SetENOAutomatically false, UDAEnableTagReadback false
   VAR
      P30x { S7_SetPoint := 'True'} : "PID_Pump2Pu1Fc";
      P120x { S7_SetPoint := 'True'} : "PID_Pump2Pu1Fc";
      P150x { S7_SetPoint := 'True'} : "PID_Pump2Pu1Fc";
      P901 { S7_SetPoint := 'True'} : "PID_Pump";
      P1301 { S7_SetPoint := 'True'} : "PID_Pump";
   END_VAR
BEGIN

REGION Network 1: P30x
